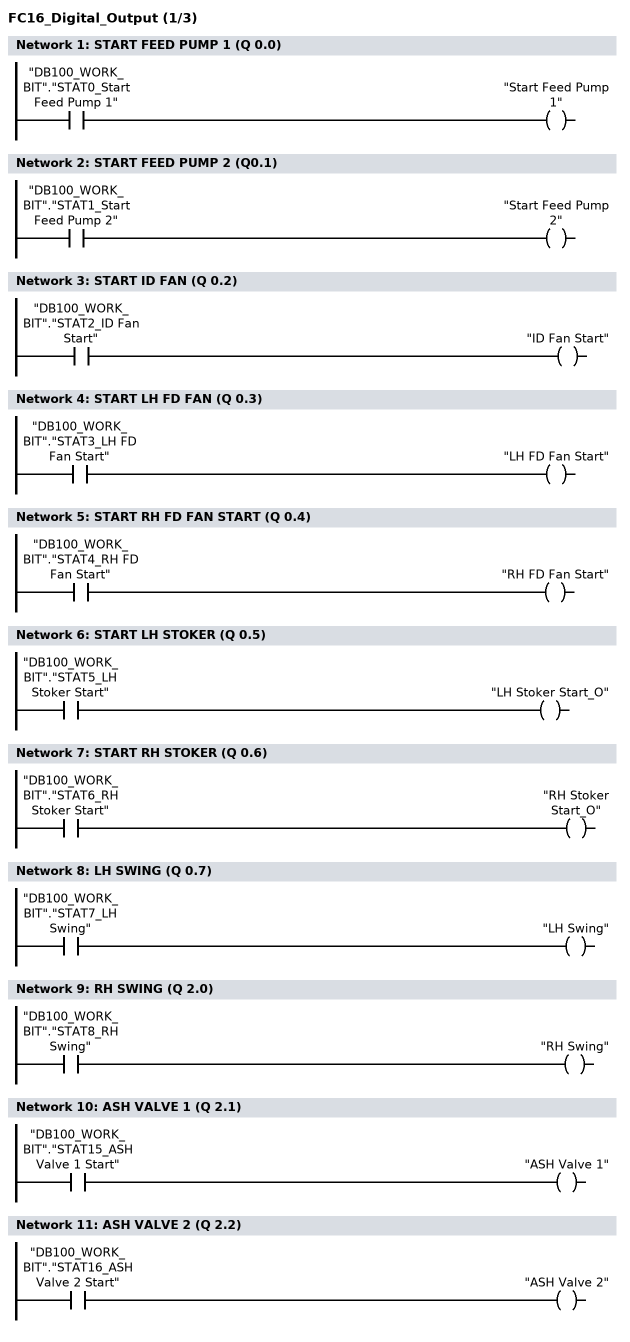
   RUNG wire#powerrail
      Contact( "DB100_WORK_BIT"."STAT0_Start Feed Pump 1" )
      Coil( "Start Feed Pump 1" )
   END_RUNG
   // the same network as SCL:
   "Start Feed Pump 1" := "DB100_WORK_BIT"."STAT0_Start Feed Pump 1";
END_REGION

REGION Network 2: START FEED PUMP 2 (Q0.1)
   RUNG wire#powerrail
      Contact( "DB100_WORK_BIT"."STAT1_Start Feed Pump 2" )
      Coil( "Start Feed Pump 2" )
   END_RUNG
   // the same network as SCL:
   "Start Feed Pump 2" := "DB100_WORK_BIT"."STAT1_Start Feed Pump 2";
END_REGION

REGION Network 3: START ID FAN (Q 0.2)
   RUNG wire#powerrail
      Contact( "DB100_WORK_BIT"."STAT2_ID Fan Start" )
      Coil( "ID Fan Start" )
   END_RUNG
   // the same network as SCL:
   "ID Fan Start" := "DB100_WORK_BIT"."STAT2_ID Fan Start";
END_REGION

REGION Network 4: START LH FD FAN (Q 0.3)
   RUNG wire#powerrail
      Contact( "DB100_WORK_BIT"."STAT3_LH FD Fan Start" )
      Coil( "LH FD Fan Start" )
   END_RUNG
   // the same network as SCL:
   "LH FD Fan Start" := "DB100_WORK_BIT"."STAT3_LH FD Fan Start";
END_REGION

REGION Network 5: START RH FD FAN START (Q 0.4)
   RUNG wire#powerrail
      Contact( "DB100_WORK_BIT"."STAT4_RH FD Fan Start" )
      Coil( "RH FD Fan Start" )
   END_RUNG
   // the same network as SCL:
   "RH FD Fan Start" := "DB100_WORK_BIT"."STAT4_RH FD Fan Start";
END_REGION

REGION Network 6: START LH STOKER (Q 0.5)
   RUNG wire#powerrail
      Contact( "DB100_WORK_BIT"."STAT5_LH Stoker Start" )
      Coil( "LH Stoker Start_O" )
   END_RUNG
   // the same network as SCL:
   "LH Stoker Start_O" := "DB100_WORK_BIT"."STAT5_LH Stoker Start";
END_REGION

REGION Network 7: START RH STOKER (Q 0.6)
   RUNG wire#powerrail
      Contact( "DB100_WORK_BIT"."STAT6_RH Stoker Start" )
      Coil( "RH Stoker Start_O" )
   END_RUNG
   // the same network as SCL:
   "RH Stoker Start_O" := "DB100_WORK_BIT"."STAT6_RH Stoker Start";
END_REGION

REGION Network 8: LH SWING (Q 0.7)
   RUNG wire#powerrail
      Contact( "DB100_WORK_BIT"."STAT7_LH Swing" )
      Coil( "LH Swing" )
   END_RUNG
   // the same network as SCL:
   "LH Swing" := "DB100_WORK_BIT"."STAT7_LH Swing";
END_REGION

REGION Network 9: RH SWING (Q 2.0)
   RUNG wire#powerrail
      Contact( "DB100_WORK_BIT"."STAT8_RH Swing" )
      Coil( "RH Swing" )
   END_RUNG
   // the same network as SCL:
   "RH Swing" := "DB100_WORK_BIT"."STAT8_RH Swing";
END_REGION

REGION Network 10: ASH VALVE 1 (Q 2.1)
   RUNG wire#powerrail
      Contact( "DB100_WORK_BIT"."STAT15_ASH Valve 1 Start" )
      Coil( "ASH Valve 1" )
   END_RUNG
   // the same network as SCL:
   "ASH Valve 1" := "DB100_WORK_BIT"."STAT15_ASH Valve 1 Start";
END_REGION

REGION Network 11: ASH VALVE 2 (Q 2.2)
   RUNG wire#powerrail
      Contact( "DB100_WORK_BIT"."STAT16_ASH Valve 2 Start" )
      Coil( "ASH Valve 2" )
   END_RUNG
   // the same network as SCL:
   "ASH Valve 2" := "DB100_WORK_BIT"."STAT16_ASH Valve 2 Start";
END_REGION

REGION Network 12: ASH CONVEYOR (Q 2.3)
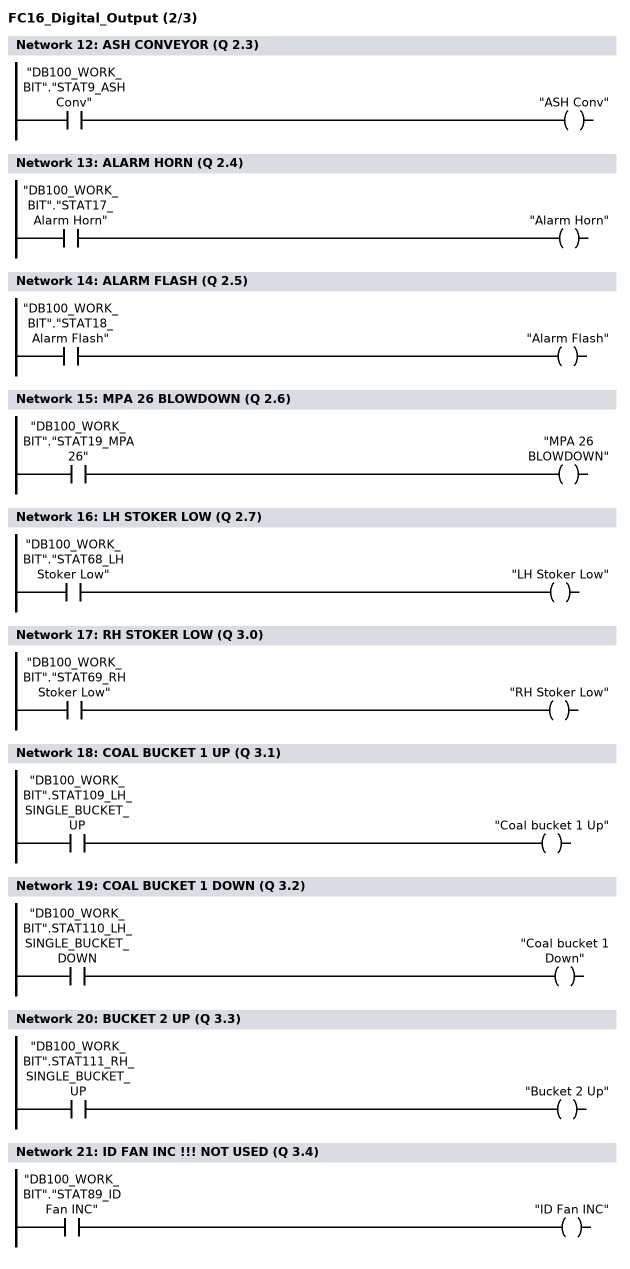
   RUNG wire#powerrail
      Contact( "DB100_WORK_BIT"."STAT9_ASH Conv" )
      Coil( "ASH Conv" )
   END_RUNG
   // the same network as SCL:
   "ASH Conv" := "DB100_WORK_BIT"."STAT9_ASH Conv";
END_REGION

REGION Network 13: ALARM HORN (Q 2.4)
   RUNG wire#powerrail
      Contact( "DB100_WORK_BIT"."STAT17_Alarm Horn" )
      Coil( "Alarm Horn" )
   END_RUNG
   // the same network as SCL:
   "Alarm Horn" := "DB100_WORK_BIT"."STAT17_Alarm Horn";
END_REGION

REGION Network 14: ALARM FLASH (Q 2.5)
   RUNG wire#powerrail
      Contact( "DB100_WORK_BIT"."STAT18_Alarm Flash" )
      Coil( "Alarm Flash" )
   END_RUNG
   // the same network as SCL:
   "Alarm Flash" := "DB100_WORK_BIT"."STAT18_Alarm Flash";
END_REGION

REGION Network 15: MPA 26 BLOWDOWN (Q 2.6)
   RUNG wire#powerrail
      Contact( "DB100_WORK_BIT"."STAT19_MPA 26" )
      Coil( "MPA 26 BLOWDOWN" )
   END_RUNG
   // the same network as SCL:
   "MPA 26 BLOWDOWN" := "DB100_WORK_BIT"."STAT19_MPA 26";
END_REGION

REGION Network 16: LH STOKER LOW (Q 2.7)
   RUNG wire#powerrail
      Contact( "DB100_WORK_BIT"."STAT68_LH Stoker Low" )
      Coil( "LH Stoker Low" )
   END_RUNG
   // the same network as SCL:
   "LH Stoker Low" := "DB100_WORK_BIT"."STAT68_LH Stoker Low";
END_REGION

REGION Network 17: RH STOKER LOW (Q 3.0)
   RUNG wire#powerrail
      Contact( "DB100_WORK_BIT"."STAT69_RH Stoker Low" )
      Coil( "RH Stoker Low" )
   END_RUNG
   // the same network as SCL:
   "RH Stoker Low" := "DB100_WORK_BIT"."STAT69_RH Stoker Low";
END_REGION

REGION Network 18: COAL BUCKET 1 UP (Q 3.1)
   RUNG wire#powerrail
      Contact( "DB100_WORK_BIT".STAT109_LH_SINGLE_BUCKET_UP )
      Coil( "Coal bucket 1 Up" )
   END_RUNG
   // the same network as SCL:
   "Coal bucket 1 Up" := "DB100_WORK_BIT".STAT109_LH_SINGLE_BUCKET_UP;
END_REGION

REGION Network 19: COAL BUCKET 1 DOWN (Q 3.2)
   RUNG wire#powerrail
      Contact( "DB100_WORK_BIT".STAT110_LH_SINGLE_BUCKET_DOWN )
      Coil( "Coal bucket 1 Down" )
   END_RUNG
   // the same network as SCL:
   "Coal bucket 1 Down" := "DB100_WORK_BIT".STAT110_LH_SINGLE_BUCKET_DOWN;
END_REGION

REGION Network 20: BUCKET 2 UP (Q 3.3)
   RUNG wire#powerrail
      Contact( "DB100_WORK_BIT".STAT111_RH_SINGLE_BUCKET_UP )
      Coil( "Bucket 2 Up" )
   END_RUNG
   // the same network as SCL:
   "Bucket 2 Up" := "DB100_WORK_BIT".STAT111_RH_SINGLE_BUCKET_UP;
END_REGION

REGION Network 21: ID FAN INC !!! NOT USED (Q 3.4)
   RUNG wire#powerrail
      Contact( "DB100_WORK_BIT"."STAT89_ID Fan INC" )
      Coil( "ID Fan INC" )
   END_RUNG
   // the same network as SCL:
   "ID Fan INC" := "DB100_WORK_BIT"."STAT89_ID Fan INC";
END_REGION

REGION Network 22: ID FAN DEC !!! NOT USED (Q 3.5)
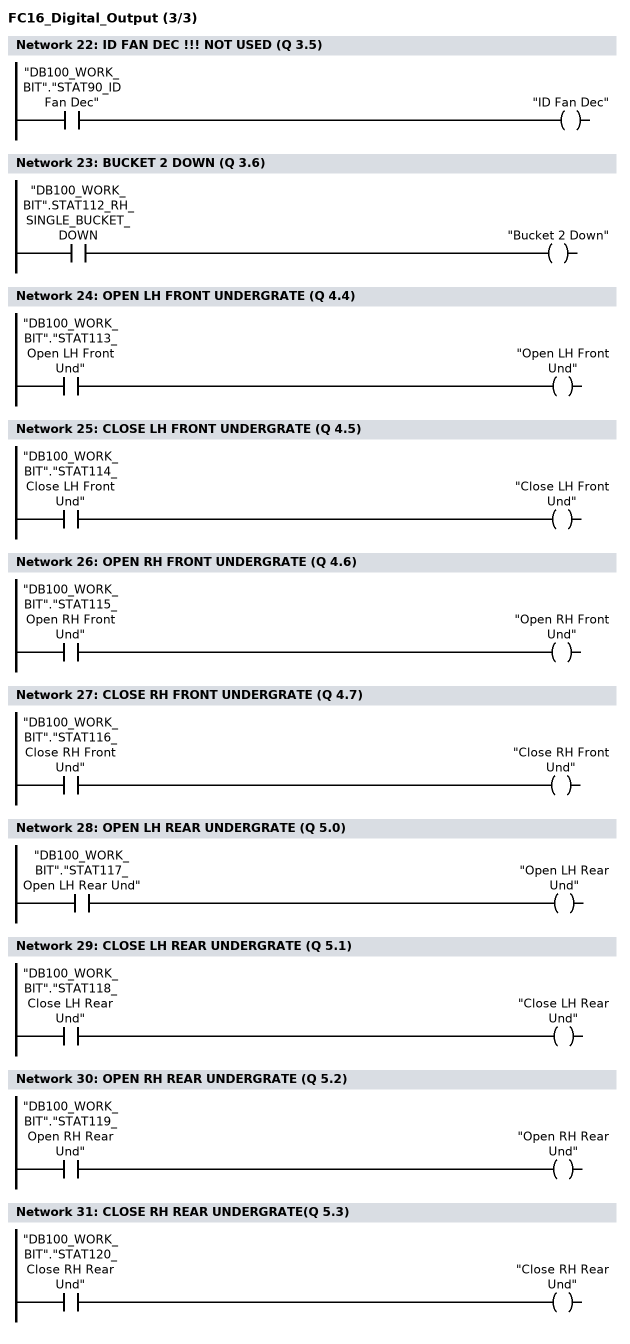
   RUNG wire#powerrail
      Contact( "DB100_WORK_BIT"."STAT90_ID Fan Dec" )
      Coil( "ID Fan Dec" )
   END_RUNG
   // the same network as SCL:
   "ID Fan Dec" := "DB100_WORK_BIT"."STAT90_ID Fan Dec";
END_REGION

REGION Network 23: BUCKET 2 DOWN (Q 3.6)
   RUNG wire#powerrail
      Contact( "DB100_WORK_BIT".STAT112_RH_SINGLE_BUCKET_DOWN )
      Coil( "Bucket 2 Down" )
   END_RUNG
   // the same network as SCL:
   "Bucket 2 Down" := "DB100_WORK_BIT".STAT112_RH_SINGLE_BUCKET_DOWN;
END_REGION

REGION Network 24: OPEN LH FRONT UNDERGRATE (Q 4.4)
   RUNG wire#powerrail
      Contact( "DB100_WORK_BIT"."STAT113_Open LH Front Und" )
      Coil( "Open LH Front Und" )
   END_RUNG
   // the same network as SCL:
   "Open LH Front Und" := "DB100_WORK_BIT"."STAT113_Open LH Front Und";
END_REGION

REGION Network 25: CLOSE LH FRONT UNDERGRATE (Q 4.5)
   RUNG wire#powerrail
      Contact( "DB100_WORK_BIT"."STAT114_Close LH Front Und" )
      Coil( "Close LH Front Und" )
   END_RUNG
   // the same network as SCL:
   "Close LH Front Und" := "DB100_WORK_BIT"."STAT114_Close LH Front Und";
END_REGION

REGION Network 26: OPEN RH FRONT UNDERGRATE (Q 4.6)
   RUNG wire#powerrail
      Contact( "DB100_WORK_BIT"."STAT115_Open RH Front Und" )
      Coil( "Open RH Front Und" )
   END_RUNG
   // the same network as SCL:
   "Open RH Front Und" := "DB100_WORK_BIT"."STAT115_Open RH Front Und";
END_REGION

REGION Network 27: CLOSE RH FRONT UNDERGRATE (Q 4.7)
   RUNG wire#powerrail
      Contact( "DB100_WORK_BIT"."STAT116_Close RH Front Und" )
      Coil( "Close RH Front Und" )
   END_RUNG
   // the same network as SCL:
   "Close RH Front Und" := "DB100_WORK_BIT"."STAT116_Close RH Front Und";
END_REGION

REGION Network 28: OPEN LH REAR UNDERGRATE (Q 5.0)
   RUNG wire#powerrail
      Contact( "DB100_WORK_BIT"."STAT117_Open LH Rear Und" )
      Coil( "Open LH Rear Und" )
   END_RUNG
   // the same network as SCL:
   "Open LH Rear Und" := "DB100_WORK_BIT"."STAT117_Open LH Rear Und";
END_REGION

REGION Network 29: CLOSE LH REAR UNDERGRATE (Q 5.1)
   RUNG wire#powerrail
      Contact( "DB100_WORK_BIT"."STAT118_Close LH Rear Und" )
      Coil( "Close LH Rear Und" )
   END_RUNG
   // the same network as SCL:
   "Close LH Rear Und" := "DB100_WORK_BIT"."STAT118_Close LH Rear Und";
END_REGION

REGION Network 30: OPEN RH REAR UNDERGRATE (Q 5.2)
   RUNG wire#powerrail
      Contact( "DB100_WORK_BIT"."STAT119_Open RH Rear Und" )
      Coil( "Open RH Rear Und" )
   END_RUNG
   // the same network as SCL:
   "Open RH Rear Und" := "DB100_WORK_BIT"."STAT119_Open RH Rear Und";
END_REGION

REGION Network 31: CLOSE RH REAR UNDERGRATE(Q 5.3)
   RUNG wire#powerrail
      Contact( "DB100_WORK_BIT"."STAT120_Close RH Rear Und" )
      Coil( "Close RH Rear Und" )
   END_RUNG
   // the same network as SCL:
   "Close RH Rear Und" := "DB100_WORK_BIT"."STAT120_Close RH Rear Und";
END_REGION
END_FUNCTION

FUNCTION "FC17_Analog_Input" : Void   // FC17, LAD
TITLE = Mapping Analog Input to DB 103
{ S7_Optimized_Access := 'TRUE' }
VERSION : 0.1
BEGIN

REGION Network 1: Pressure Transducer IW 100
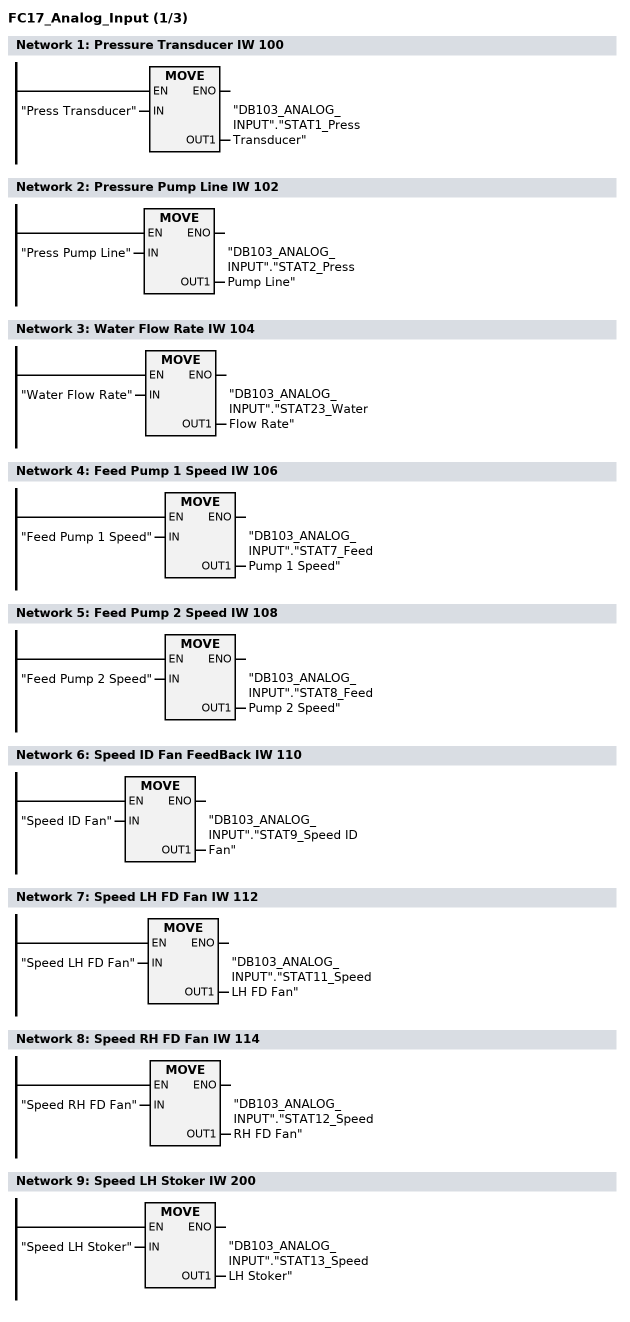
   RUNG wire#powerrail
      Move(in := "Press Transducer", out1 => "DB103_ANALOG_INPUT"."STAT1_Press Transducer")
   END_RUNG
   // the same network as SCL:
   "DB103_ANALOG_INPUT"."STAT1_Press Transducer" := "Press Transducer";
END_REGION

REGION Network 2: Pressure Pump Line IW 102
   RUNG wire#powerrail
      Move(in := "Press Pump Line", out1 => "DB103_ANALOG_INPUT"."STAT2_Press Pump Line")
   END_RUNG
   // the same network as SCL:
   "DB103_ANALOG_INPUT"."STAT2_Press Pump Line" := "Press Pump Line";
END_REGION

REGION Network 3: Water Flow Rate IW 104
   RUNG wire#powerrail
      Move(in := "Water Flow Rate", out1 => "DB103_ANALOG_INPUT"."STAT23_Water Flow Rate")
   END_RUNG
   // the same network as SCL:
   "DB103_ANALOG_INPUT"."STAT23_Water Flow Rate" := "Water Flow Rate";
END_REGION

REGION Network 4: Feed Pump 1 Speed IW 106
   RUNG wire#powerrail
      Move(in := "Feed Pump 1 Speed", out1 => "DB103_ANALOG_INPUT"."STAT7_Feed Pump 1 Speed")
   END_RUNG
   // the same network as SCL:
   "DB103_ANALOG_INPUT"."STAT7_Feed Pump 1 Speed" := "Feed Pump 1 Speed";
END_REGION

REGION Network 5: Feed Pump 2 Speed IW 108
   RUNG wire#powerrail
      Move(in := "Feed Pump 2 Speed", out1 => "DB103_ANALOG_INPUT"."STAT8_Feed Pump 2 Speed")
   END_RUNG
   // the same network as SCL:
   "DB103_ANALOG_INPUT"."STAT8_Feed Pump 2 Speed" := "Feed Pump 2 Speed";
END_REGION

REGION Network 6: Speed ID Fan FeedBack IW 110
   RUNG wire#powerrail
      Move(in := "Speed ID Fan", out1 => "DB103_ANALOG_INPUT"."STAT9_Speed ID Fan")
   END_RUNG
   // the same network as SCL:
   "DB103_ANALOG_INPUT"."STAT9_Speed ID Fan" := "Speed ID Fan";
END_REGION

REGION Network 7: Speed LH FD Fan IW 112
   RUNG wire#powerrail
      Move(in := "Speed LH FD Fan", out1 => "DB103_ANALOG_INPUT"."STAT11_Speed LH FD Fan")
   END_RUNG
   // the same network as SCL:
   "DB103_ANALOG_INPUT"."STAT11_Speed LH FD Fan" := "Speed LH FD Fan";
END_REGION

REGION Network 8: Speed RH FD Fan IW 114
   RUNG wire#powerrail
      Move(in := "Speed RH FD Fan", out1 => "DB103_ANALOG_INPUT"."STAT12_Speed RH FD Fan")
   END_RUNG
   // the same network as SCL:
   "DB103_ANALOG_INPUT"."STAT12_Speed RH FD Fan" := "Speed RH FD Fan";
END_REGION

REGION Network 9: Speed LH Stoker IW 200
   RUNG wire#powerrail
      Move(in := "Speed LH Stoker", out1 => "DB103_ANALOG_INPUT"."STAT13_Speed LH Stoker")
   END_RUNG
   // the same network as SCL:
   "DB103_ANALOG_INPUT"."STAT13_Speed LH Stoker" := "Speed LH Stoker";
END_REGION

REGION Network 10: Speed RH Stoker IW 202
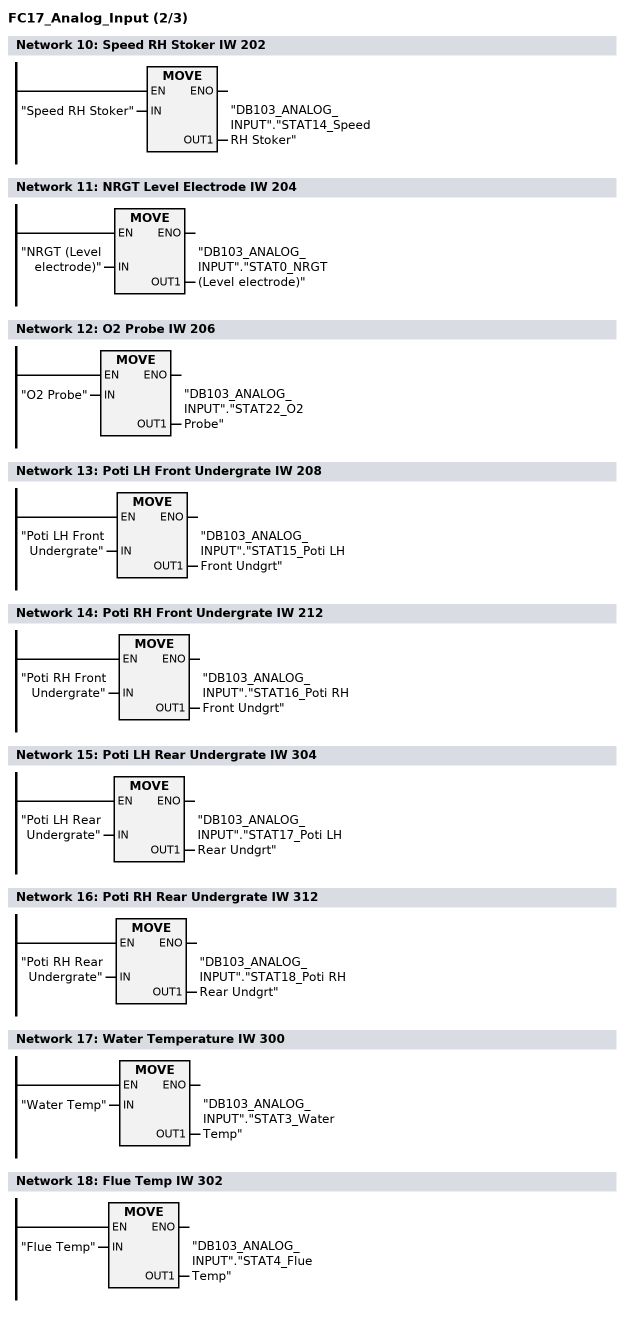
   RUNG wire#powerrail
      Move(in := "Speed RH Stoker", out1 => "DB103_ANALOG_INPUT"."STAT14_Speed RH Stoker")
   END_RUNG
   // the same network as SCL:
   "DB103_ANALOG_INPUT"."STAT14_Speed RH Stoker" := "Speed RH Stoker";
END_REGION

REGION Network 11: NRGT Level Electrode IW 204
   RUNG wire#powerrail
      Move(in := "NRGT (Level electrode)", out1 => "DB103_ANALOG_INPUT"."STAT0_NRGT (Level electrode)")
   END_RUNG
   // the same network as SCL:
   "DB103_ANALOG_INPUT"."STAT0_NRGT (Level electrode)" := "NRGT (Level electrode)";
END_REGION

REGION Network 12: O2 Probe IW 206
   RUNG wire#powerrail
      Move(in := "O2 Probe", out1 => "DB103_ANALOG_INPUT"."STAT22_O2 Probe")
   END_RUNG
   // the same network as SCL:
   "DB103_ANALOG_INPUT"."STAT22_O2 Probe" := "O2 Probe";
END_REGION

REGION Network 13: Poti LH Front Undergrate IW 208
   RUNG wire#powerrail
      Move(in := "Poti LH Front Undergrate", out1 => "DB103_ANALOG_INPUT"."STAT15_Poti LH Front Undgrt")
   END_RUNG
   // the same network as SCL:
   "DB103_ANALOG_INPUT"."STAT15_Poti LH Front Undgrt" := "Poti LH Front Undergrate";
END_REGION

REGION Network 14: Poti RH Front Undergrate IW 212
   RUNG wire#powerrail
      Move(in := "Poti RH Front Undergrate", out1 => "DB103_ANALOG_INPUT"."STAT16_Poti RH Front Undgrt")
   END_RUNG
   // the same network as SCL:
   "DB103_ANALOG_INPUT"."STAT16_Poti RH Front Undgrt" := "Poti RH Front Undergrate";
END_REGION

REGION Network 15: Poti LH Rear Undergrate IW 304
   RUNG wire#powerrail
      Move(in := "Poti LH Rear Undergrate", out1 => "DB103_ANALOG_INPUT"."STAT17_Poti LH Rear Undgrt")
   END_RUNG
   // the same network as SCL:
   "DB103_ANALOG_INPUT"."STAT17_Poti LH Rear Undgrt" := "Poti LH Rear Undergrate";
END_REGION

REGION Network 16: Poti RH Rear Undergrate IW 312
   RUNG wire#powerrail
      Move(in := "Poti RH Rear Undergrate", out1 => "DB103_ANALOG_INPUT"."STAT18_Poti RH Rear Undgrt")
   END_RUNG
   // the same network as SCL:
   "DB103_ANALOG_INPUT"."STAT18_Poti RH Rear Undgrt" := "Poti RH Rear Undergrate";
END_REGION

REGION Network 17: Water Temperature IW 300
   RUNG wire#powerrail
      Move(in := "Water Temp", out1 => "DB103_ANALOG_INPUT"."STAT3_Water Temp")
   END_RUNG
   // the same network as SCL:
   "DB103_ANALOG_INPUT"."STAT3_Water Temp" := "Water Temp";
END_REGION

REGION Network 18: Flue Temp IW 302
   RUNG wire#powerrail
      Move(in := "Flue Temp", out1 => "DB103_ANALOG_INPUT"."STAT4_Flue Temp")
   END_RUNG
   // the same network as SCL:
   "DB103_ANALOG_INPUT"."STAT4_Flue Temp" := "Flue Temp";
END_REGION

REGION Network 19: LH Thermocouple IW 308
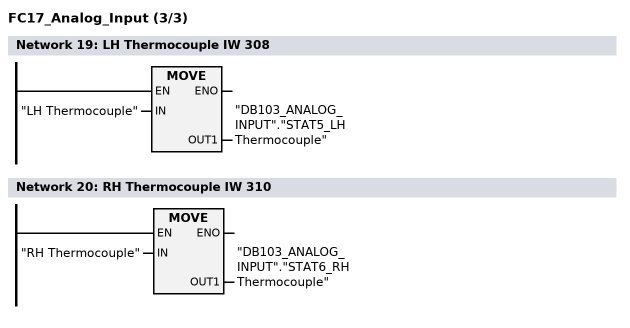
   RUNG wire#powerrail
      Move(in := "LH Thermocouple", out1 => "DB103_ANALOG_INPUT"."STAT5_LH Thermocouple")
   END_RUNG
   // the same network as SCL:
   "DB103_ANALOG_INPUT"."STAT5_LH Thermocouple" := "LH Thermocouple";
END_REGION

REGION Network 20: RH Thermocouple IW 310
   RUNG wire#powerrail
      Move(in := "RH Thermocouple", out1 => "DB103_ANALOG_INPUT"."STAT6_RH Thermocouple")
   END_RUNG
   // the same network as SCL:
   "DB103_ANALOG_INPUT"."STAT6_RH Thermocouple" := "RH Thermocouple";
END_REGION
END_FUNCTION

FUNCTION "FC18_Analog_Output" : Void   // FC18, LAD
TITLE = Mapping Analog Output from DB 140
{ S7_Optimized_Access := 'TRUE' }
VERSION : 0.1
BEGIN

REGION Network 1: Feed Pump 1 Reference Speed QW 500
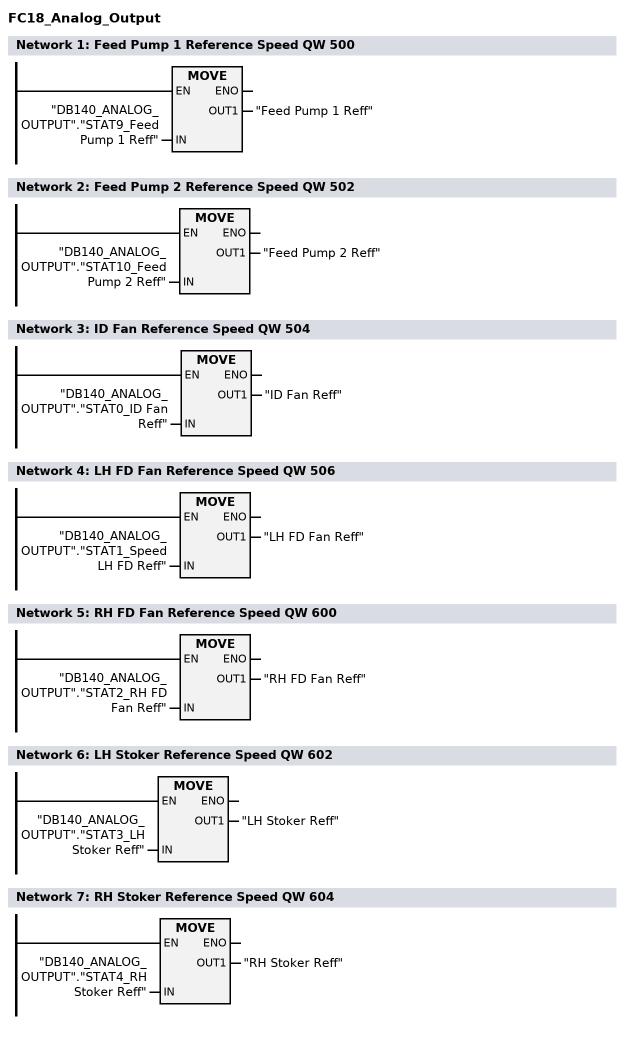
   RUNG wire#powerrail
      Move(in := "DB140_ANALOG_OUTPUT"."STAT9_Feed Pump 1 Reff", out1 => "Feed Pump 1 Reff")
   END_RUNG
   // the same network as SCL:
   "Feed Pump 1 Reff" := "DB140_ANALOG_OUTPUT"."STAT9_Feed Pump 1 Reff";
END_REGION

REGION Network 2: Feed Pump 2 Reference Speed QW 502
   RUNG wire#powerrail
      Move(in := "DB140_ANALOG_OUTPUT"."STAT10_Feed Pump 2 Reff", out1 => "Feed Pump 2 Reff")
   END_RUNG
   // the same network as SCL:
   "Feed Pump 2 Reff" := "DB140_ANALOG_OUTPUT"."STAT10_Feed Pump 2 Reff";
END_REGION

REGION Network 3: ID Fan Reference Speed QW 504
   RUNG wire#powerrail
      Move(in := "DB140_ANALOG_OUTPUT"."STAT0_ID Fan Reff", out1 => "ID Fan Reff")
   END_RUNG
   // the same network as SCL:
   "ID Fan Reff" := "DB140_ANALOG_OUTPUT"."STAT0_ID Fan Reff";
END_REGION

REGION Network 4: LH FD Fan Reference Speed QW 506
   RUNG wire#powerrail
      Move(in := "DB140_ANALOG_OUTPUT"."STAT1_Speed LH FD Reff", out1 => "LH FD Fan Reff")
   END_RUNG
   // the same network as SCL:
   "LH FD Fan Reff" := "DB140_ANALOG_OUTPUT"."STAT1_Speed LH FD Reff";
END_REGION

REGION Network 5: RH FD Fan Reference Speed QW 600
   RUNG wire#powerrail
      Move(in := "DB140_ANALOG_OUTPUT"."STAT2_RH FD Fan Reff", out1 => "RH FD Fan Reff")
   END_RUNG
   // the same network as SCL:
   "RH FD Fan Reff" := "DB140_ANALOG_OUTPUT"."STAT2_RH FD Fan Reff";
END_REGION

REGION Network 6: LH Stoker Reference Speed QW 602
   RUNG wire#powerrail
      Move(in := "DB140_ANALOG_OUTPUT"."STAT3_LH Stoker Reff", out1 => "LH Stoker Reff")
   END_RUNG
   // the same network as SCL:
   "LH Stoker Reff" := "DB140_ANALOG_OUTPUT"."STAT3_LH Stoker Reff";
END_REGION

REGION Network 7: RH Stoker Reference Speed QW 604
   RUNG wire#powerrail
      Move(in := "DB140_ANALOG_OUTPUT"."STAT4_RH Stoker Reff", out1 => "RH Stoker Reff")
   END_RUNG
   // the same network as SCL:
   "RH Stoker Reff" := "DB140_ANALOG_OUTPUT"."STAT4_RH Stoker Reff";
END_REGION
END_FUNCTION

FUNCTION "FC105_scalling AI" : Void   // FC105, LAD
TITLE = SCALLING ANALOG INPUT
{ S7_Optimized_Access := 'TRUE' }
VERSION : 0.1
// rumus scalling
// 
// norm_x  = out =  (VALUE – MIN) / (MAX – MIN)
// scale_x  = out =( (max-min)*value)+min
   VAR_INPUT
      IN0 : Int;
      IN1 : Real;
      IN2 : Real;
      IN3 : Bool;
   END_VAR
   VAR_OUTPUT
      Out4 : Real;
      RET_VAL_1 : Word;
   END_VAR
   VAR_TEMP
      Temp5 : Real;
      Temp6 : Real;
      Temp7 : Real;
      Temp8 : Real;
      Temp9 : Real;
      Temp10 : DInt;
      Temp11 : Bool;
      Temp12 : Bool;
      Temp13 : Real;
      Temp14 : Real;
      Temp15 : Real;
   END_VAR
   VAR_TEMP   // added for the SCL form of the ladder/FBD networks
      _w1 : Bool;
   END_VAR
BEGIN

REGION Network 1: K1 min
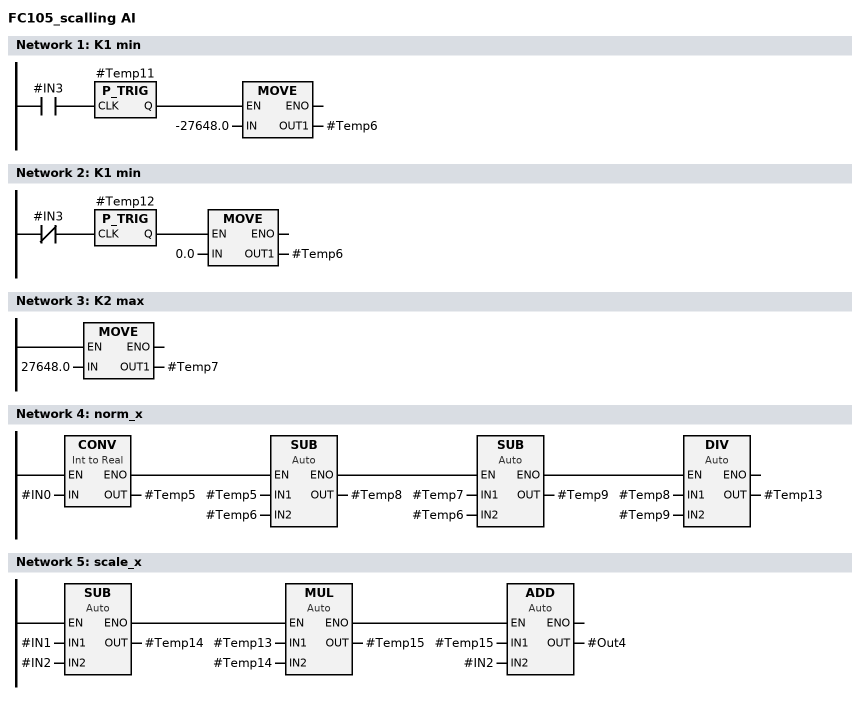
   RUNG wire#powerrail
      Contact( #IN3 )
      P_Trig( #Temp11 )
      Move(in := -27648.0, out1 => #Temp6)
   END_RUNG
   // the same network as SCL:
   #_w1 := #IN3 AND NOT #Temp11;   // rising edge
   #Temp11 := #IN3;
   IF #_w1 THEN #Temp6 := -27648.0; END_IF;
END_REGION

REGION Network 2: K1 min
   RUNG wire#powerrail
      I_Contact( #IN3 )
      P_Trig( #Temp12 )
      Move(in := 0.0, out1 => #Temp6)
   END_RUNG
   // the same network as SCL:
   #_w1 := NOT #IN3 AND NOT #Temp12;   // rising edge
   #Temp12 := NOT #IN3;
   IF #_w1 THEN #Temp6 := 0.0; END_IF;
END_REGION

REGION Network 3: K2 max
   RUNG wire#powerrail
      Move(in := 27648.0, out1 => #Temp7)
   END_RUNG
   // the same network as SCL:
   #Temp7 := 27648.0;
END_REGION

REGION Network 4: norm_x
   RUNG wire#powerrail
      { S7_Templates := "[SrcType := Int, DestType := Real]" } Convert(in := #IN0, out => #Temp5)
      Sub(in1 := #Temp5, in2 := #Temp6, out => #Temp8)
      Sub(in1 := #Temp7, in2 := #Temp6, out => #Temp9)
      Div(in1 := #Temp8, in2 := #Temp9, out => #Temp13)
   END_RUNG
   // the same network as SCL:
   #Temp5 := INT_TO_REAL(#IN0);
   #Temp8 := #Temp5 - #Temp6;
   #Temp9 := #Temp7 - #Temp6;
   #Temp13 := #Temp8 / #Temp9;
END_REGION

REGION Network 5: scale_x
   RUNG wire#powerrail
      Sub(in1 := #IN1, in2 := #IN2, out => #Temp14)
      Mul(in1 := #Temp13, in2 := #Temp14, out => #Temp15)
      Add(in1 := #Temp15, in2 := #IN2, out => #Out4)
   END_RUNG
   // the same network as SCL:
   #Temp14 := #IN1 - #IN2;
   #Temp15 := #Temp13 * #Temp14;
   #Out4 := #Temp15 + #IN2;
END_REGION
END_FUNCTION

FUNCTION "FC106_Unscalling" : Void   // FC106, LAD
TITLE = UNSCALLING
{ S7_Optimized_Access := 'TRUE' }
VERSION : 0.1
// rumus scalling
// 
// norm_x  = out =  (VALUE – MIN) / (MAX – MIN)
// scale_x  = out =( (max-min)*value)+min
   VAR_INPUT
      IN0 : Real;
      IN1 : Real;
      IN2 : Real;
      IN3 : Bool;
   END_VAR
   VAR_OUTPUT
      Out4 : Int;
   END_VAR
   VAR_TEMP
      Temp5 : Real;
      Temp6 : Real;
      Temp7 : Real;
      Temp8 : Real;
      Temp9 : Real;
      Temp10 : Real;
      Temp11 : Bool;
      Temp12 : Bool;
      Temp13 : Real;
      Temp14 : Real;
      Temp15 : Int;
   END_VAR
   VAR_TEMP   // added for the SCL form of the ladder/FBD networks
      _w1 : Bool;
   END_VAR
BEGIN

REGION Network 1: MIN
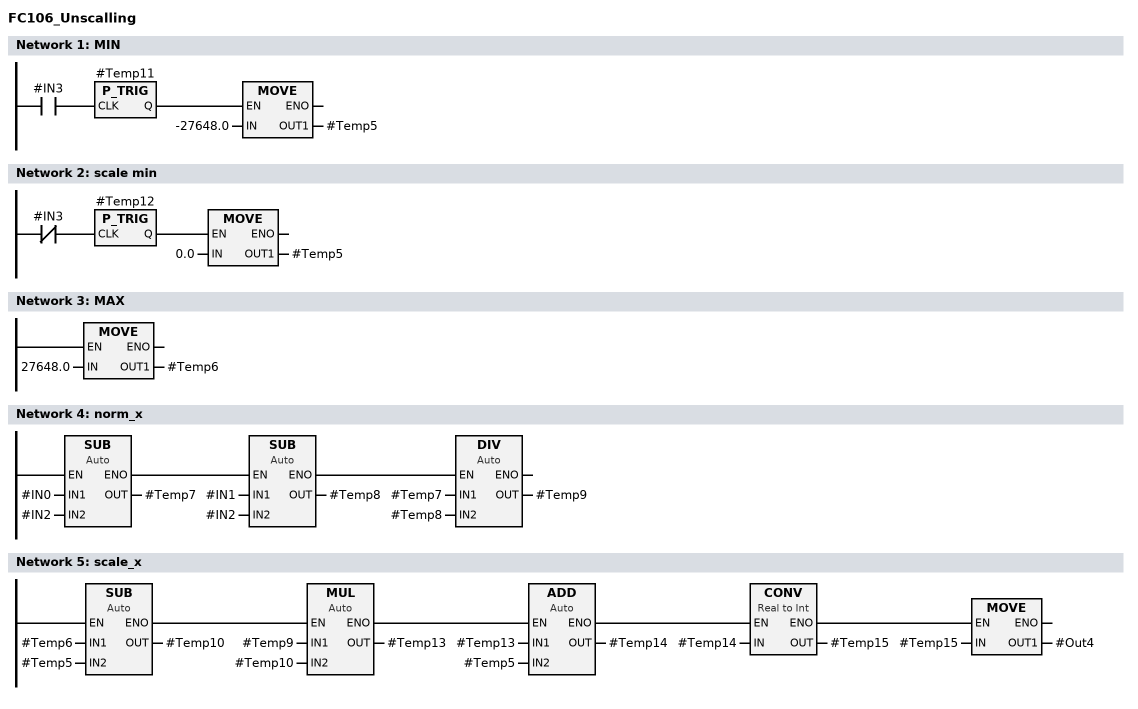
   RUNG wire#powerrail
      Contact( #IN3 )
      P_Trig( #Temp11 )
      Move(in := -27648.0, out1 => #Temp5)
   END_RUNG
   // the same network as SCL:
   #_w1 := #IN3 AND NOT #Temp11;   // rising edge
   #Temp11 := #IN3;
   IF #_w1 THEN #Temp5 := -27648.0; END_IF;
END_REGION

REGION Network 2: scale min
   RUNG wire#powerrail
      I_Contact( #IN3 )
      P_Trig( #Temp12 )
      Move(in := 0.0, out1 => #Temp5)
   END_RUNG
   // the same network as SCL:
   #_w1 := NOT #IN3 AND NOT #Temp12;   // rising edge
   #Temp12 := NOT #IN3;
   IF #_w1 THEN #Temp5 := 0.0; END_IF;
END_REGION

REGION Network 3: MAX
   RUNG wire#powerrail
      Move(in := 27648.0, out1 => #Temp6)
   END_RUNG
   // the same network as SCL:
   #Temp6 := 27648.0;
END_REGION

REGION Network 4: norm_x
   RUNG wire#powerrail
      Sub(in1 := #IN0, in2 := #IN2, out => #Temp7)
      Sub(in1 := #IN1, in2 := #IN2, out => #Temp8)
      Div(in1 := #Temp7, in2 := #Temp8, out => #Temp9)
   END_RUNG
   // the same network as SCL:
   #Temp7 := #IN0 - #IN2;
   #Temp8 := #IN1 - #IN2;
   #Temp9 := #Temp7 / #Temp8;
END_REGION

REGION Network 5: scale_x
   RUNG wire#powerrail
      Sub(in1 := #Temp6, in2 := #Temp5, out => #Temp10)
      Mul(in1 := #Temp9, in2 := #Temp10, out => #Temp13)
      Add(in1 := #Temp13, in2 := #Temp5, out => #Temp14)
      { S7_Templates := "[SrcType := Real, DestType := Int]" } Convert(in := #Temp14, out => #Temp15)
      Move(in := #Temp15, out1 => #Out4)
   END_RUNG
   // the same network as SCL:
   #Temp10 := #Temp6 - #Temp5;
   #Temp13 := #Temp9 * #Temp10;
   #Temp14 := #Temp13 + #Temp5;
   #Temp15 := REAL_TO_INT(#Temp14);
   #Out4 := #Temp15;
END_REGION
END_FUNCTION

FUNCTION "FC108_Unscalling_Custom" : Void   // FC108, LAD
TITLE = UNSCALLING CUSTOM
{ S7_Optimized_Access := 'TRUE' }
VERSION : 0.1
   VAR_INPUT
      IN0 : Real;
      IN1 : Real;
      IN2 : Real;
      IN3 : Bool;
      IN4 : Real;
      IN5 : Real;
   END_VAR
   VAR_OUTPUT
      OUT_4 : Int;
   END_VAR
   VAR_TEMP
      TEMP_7 : Int;
      TEMP_8 : Int;
      TEMP_9 : Real;
   END_VAR
BEGIN

REGION Network 1: IN4 = MIN , IN5 = MAX
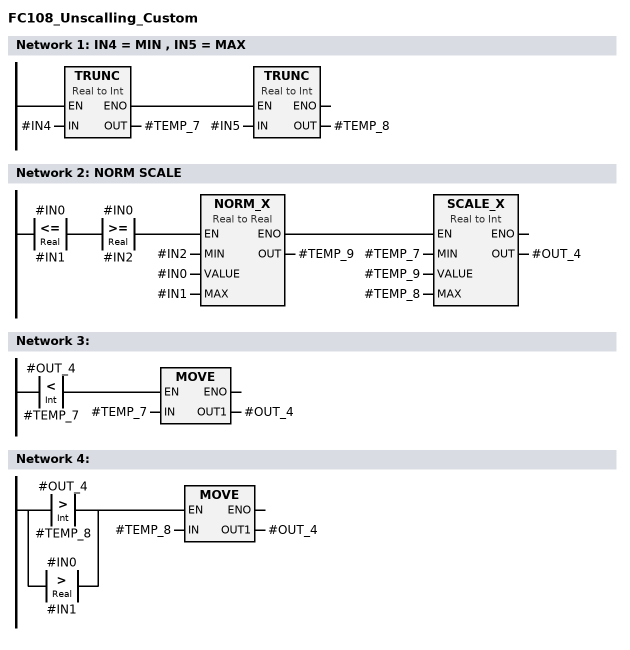
   RUNG wire#powerrail
      { S7_Templates := "[SrcType := Real, DestType := Int]" } Trunc(in := #IN4, out => #TEMP_7)
      { S7_Templates := "[SrcType := Real, DestType := Int]" } Trunc(in := #IN5, out => #TEMP_8)
   END_RUNG
   // the same network as SCL:
   #TEMP_7 := TRUNC(#IN4);
   #TEMP_8 := TRUNC(#IN5);
END_REGION

REGION Network 2: NORM SCALE
   RUNG wire#powerrail
      { S7_Templates := "SrcType := Real" } LE_Contact(in1 := #IN0, in2 := #IN1)
      { S7_Templates := "SrcType := Real" } GE_Contact(in1 := #IN0, in2 := #IN2)
      { S7_Templates := "[SrcType := Real, DestType := Real]" } Normalize(min := #IN2, value := #IN0, max := #IN1, out => #TEMP_9)
      { S7_Templates := "[SrcType := Real, DestType := Int]" } Scale(min := #TEMP_7, value := #TEMP_9, max := #TEMP_8, out => #OUT_4)
   END_RUNG
   // the same network as SCL:
   IF (#IN0 <= #IN1) AND (#IN0 >= #IN2) THEN
       #TEMP_9 := NORM_X(MIN := #IN2, VALUE := #IN0, MAX := #IN1);
       #OUT_4 := SCALE_X(MIN := #TEMP_7, VALUE := #TEMP_9, MAX := #TEMP_8);
   END_IF;
END_REGION

REGION Network 3
   RUNG wire#powerrail
      { S7_Templates := "SrcType := Int" } LT_Contact(in1 := #OUT_4, in2 := #TEMP_7)
      Move(in := #TEMP_7, out1 => #OUT_4)
   END_RUNG
   // the same network as SCL:
   IF #OUT_4 < #TEMP_7 THEN #OUT_4 := #TEMP_7; END_IF;
END_REGION

REGION Network 4
   RUNG wire#powerrail
      { S7_Templates := "SrcType := Int" } GT_Contact(in1 := #OUT_4, in2 := #TEMP_8)
      wire#w1
      Move(in := #TEMP_8, out1 => #OUT_4)
   END_RUNG
   RUNG wire#powerrail
      { S7_Templates := "SrcType := Real" } GT_Contact(in1 := #IN0, in2 := #IN1)
   END_RUNG wire#w1
   // the same network as SCL:
   IF (#OUT_4 > #TEMP_8) OR (#IN0 > #IN1) THEN #OUT_4 := #TEMP_8; END_IF;
END_REGION
END_FUNCTION

FUNCTION "FC109_Scalling_AI_Custom" : Void   // FC109, LAD
TITLE = SCALLING AI CUSTOM
{ S7_Optimized_Access := 'TRUE' }
VERSION : 0.1
// For analog in undergrate damper
   VAR_INPUT
      IN0 : Int;
      IN1 : Real;
      IN2 : Real;
      IN3 : Bool;
      IN4 : Real;
      IN5 : Real;
   END_VAR
   VAR_OUTPUT
      Out4 : Real;
      RET_VAL_1 : Word;
   END_VAR
   VAR_TEMP
      TEMP_8 : Int;
      TEMP_7 : Int;
      TEMP_9 : Real;
      TEMP_10 : Real;
   END_VAR
BEGIN

REGION Network 1: convert integer to real
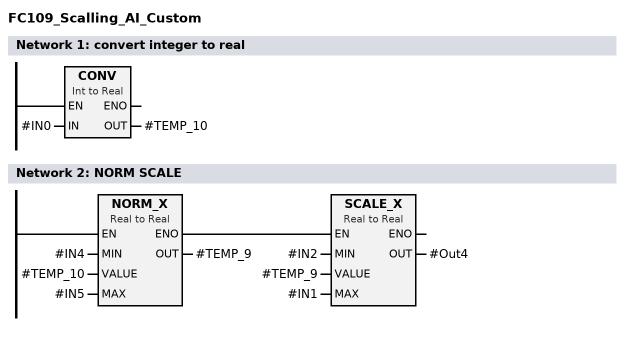
   RUNG wire#powerrail
      { S7_Templates := "[SrcType := Int, DestType := Real]" } Convert(in := #IN0, out => #TEMP_10)
   END_RUNG
   // the same network as SCL:
   #TEMP_10 := INT_TO_REAL(#IN0);
END_REGION

REGION Network 2: NORM SCALE
   RUNG wire#powerrail
      { S7_Templates := "[SrcType := Real, DestType := Real]" } Normalize(min := #IN4, value := #TEMP_10, max := #IN5, out => #TEMP_9)
      { S7_Templates := "[SrcType := Real, DestType := Real]" } Scale(min := #IN2, value := #TEMP_9, max := #IN1, out => #Out4)
   END_RUNG
   // the same network as SCL:
   #TEMP_9 := NORM_X(MIN := #IN4, VALUE := #TEMP_10, MAX := #IN5);
   #Out4 := SCALE_X(MIN := #IN2, VALUE := #TEMP_9, MAX := #IN1);
END_REGION
END_FUNCTION

FUNCTION "FC110_GENERAL_BIT" : Void   // FC110, LAD
{ S7_Optimized_Access := 'TRUE' }
VERSION : 0.1
BEGIN

REGION Network 1: Always TRUE
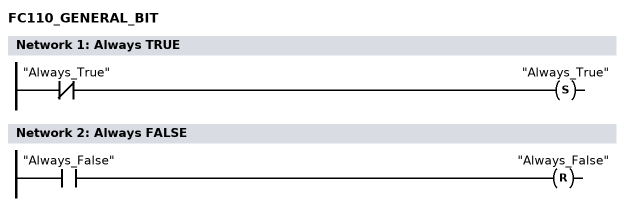
   RUNG wire#powerrail
      I_Contact( "Always_True" )
      S_Coil( "Always_True" )
   END_RUNG
   // the same network as SCL:
   IF NOT "Always_True" THEN "Always_True" := TRUE; END_IF;
END_REGION

REGION Network 2: Always FALSE
   RUNG wire#powerrail
      Contact( "Always_False" )
      R_Coil( "Always_False" )
   END_RUNG
   // the same network as SCL:
   IF "Always_False" THEN "Always_False" := FALSE; END_IF;
END_REGION
END_FUNCTION

FUNCTION "FC112_DATE_TIME" : Void   // FC112, LAD
TITLE = DATE TIME PLC SETTING
{ S7_Optimized_Access := 'TRUE' }
VERSION : 0.1
   VAR_TEMP
      v1 : Int;
      v2 : Word;
      v3 : Int;
      v4 : Word;
      v5 : Int;
      v6 : Word;
      v7 : Int;
      v8 : Word;
      v9 : Int;
      v10 : String;
      v11 : String;
      v12 : Int;
      v13 : Int;
      v14 : Word;
      v15 : Int;
      v16 : Word;
      v17 : Int;
      v18 : Word;
   END_VAR
   VAR_TEMP   // added for the SCL form of the ladder/FBD networks
      _w1 : Bool;
   END_VAR
BEGIN

REGION Network 1: READ DATE TIME
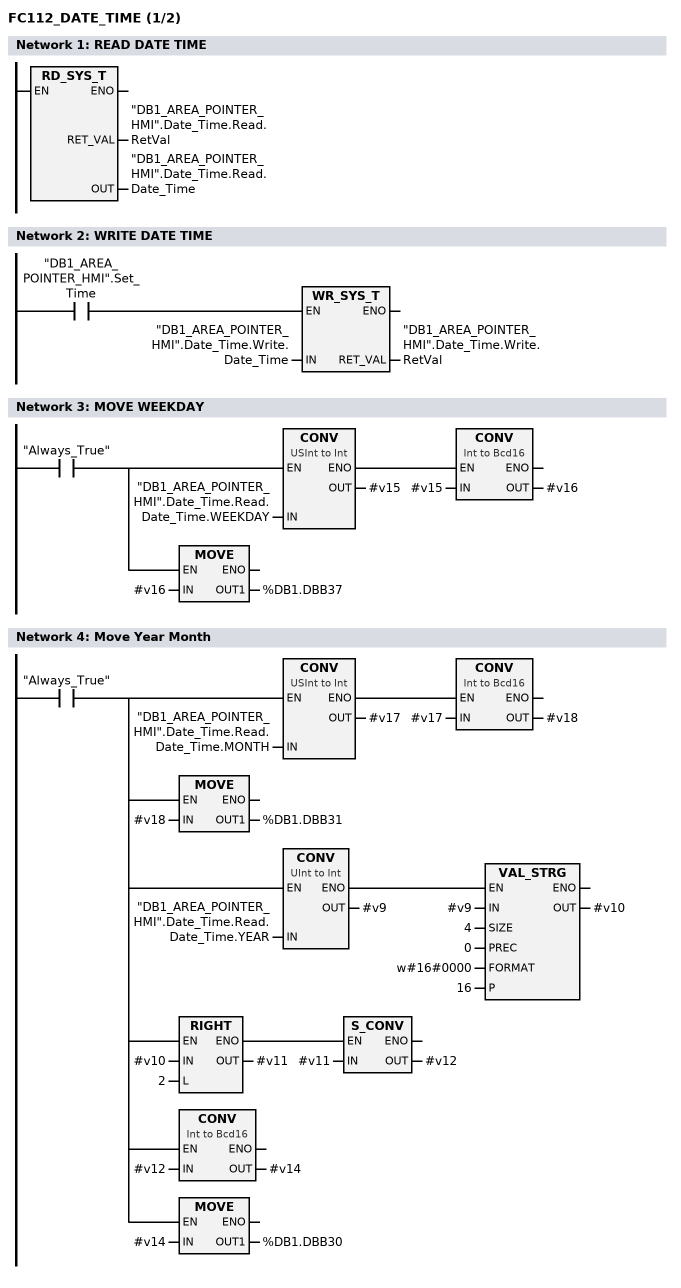
   "DB1_AREA_POINTER_HMI".Date_Time.Read.RetVal := RD_SYS_T(OUT => "DB1_AREA_POINTER_HMI".Date_Time.Read.Date_Time);
END_REGION

REGION Network 2: WRITE DATE TIME
   IF "DB1_AREA_POINTER_HMI".Set_Time THEN
       "DB1_AREA_POINTER_HMI".Date_Time.Write.RetVal := WR_SYS_T(IN := "DB1_AREA_POINTER_HMI".Date_Time.Write.Date_Time);
   END_IF;
END_REGION

REGION Network 3: MOVE WEEKDAY
   RUNG wire#powerrail
      Contact( "Always_True" )
      wire#w1
      { S7_Templates := "[SrcType := USInt, DestType := Int]" } Convert(in := "DB1_AREA_POINTER_HMI".Date_Time.Read.Date_Time.WEEKDAY, out => #v15)
      { S7_Templates := "[SrcType := Int, DestType := Bcd16]" } Convert(in := #v15, out => #v16)
   END_RUNG
   RUNG wire#w1
      Move(in := #v16, out1 => %DB1.DBB37)
   END_RUNG
   // the same network as SCL:
   IF "Always_True" THEN
       #v15 := USINT_TO_INT("DB1_AREA_POINTER_HMI".Date_Time.Read.Date_Time.WEEKDAY);
       #v16 := INT_TO_BCD16(#v15);
       %DB1.DBB37 := #v16;
   END_IF;
END_REGION

REGION Network 4: Move Year Month
   IF "Always_True" THEN
       #v17 := USINT_TO_INT("DB1_AREA_POINTER_HMI".Date_Time.Read.Date_Time.MONTH);
       #v18 := INT_TO_BCD16(#v17);
       %DB1.DBB31 := #v18;
       #v9 := UINT_TO_INT("DB1_AREA_POINTER_HMI".Date_Time.Read.Date_Time.YEAR);
   END_IF;
   #_w1 := "Always_True";
   IF #_w1 THEN
       VAL_STRG(IN := #v9, SIZE := 4, PREC := 0, FORMAT := w#16#0000, P := 16, OUT => #v10);
       #v11 := RIGHT(IN := #v10, L := 2);
       #v12 := S_CONV(IN := #v11);
       #v14 := INT_TO_BCD16(#v12);
       %DB1.DBB30 := #v14;
   END_IF;
END_REGION

REGION Network 5: Move Day &Hour
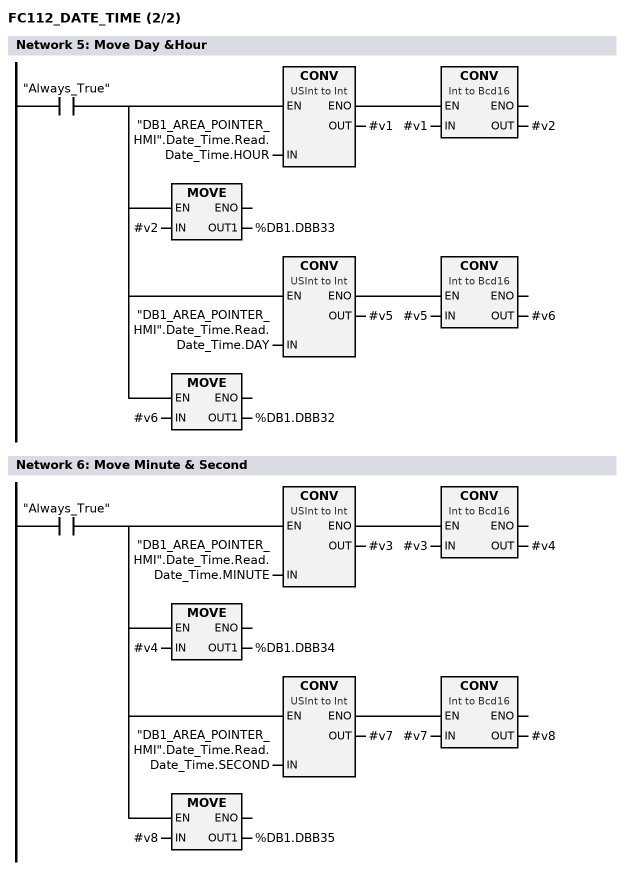
   RUNG wire#powerrail
      Contact( "Always_True" )
      wire#w1
      { S7_Templates := "[SrcType := USInt, DestType := Int]" } Convert(in := "DB1_AREA_POINTER_HMI".Date_Time.Read.Date_Time.HOUR, out => #v1)
      { S7_Templates := "[SrcType := Int, DestType := Bcd16]" } Convert(in := #v1, out => #v2)
   END_RUNG
   RUNG wire#w1
      Move(in := #v2, out1 => %DB1.DBB33)
   END_RUNG
   RUNG wire#w1
      { S7_Templates := "[SrcType := USInt, DestType := Int]" } Convert(in := "DB1_AREA_POINTER_HMI".Date_Time.Read.Date_Time.DAY, out => #v5)
      { S7_Templates := "[SrcType := Int, DestType := Bcd16]" } Convert(in := #v5, out => #v6)
   END_RUNG
   RUNG wire#w1
      Move(in := #v6, out1 => %DB1.DBB32)
   END_RUNG
   // the same network as SCL:
   IF "Always_True" THEN
       #v1 := USINT_TO_INT("DB1_AREA_POINTER_HMI".Date_Time.Read.Date_Time.HOUR);
       #v2 := INT_TO_BCD16(#v1);
       %DB1.DBB33 := #v2;
       #v5 := USINT_TO_INT("DB1_AREA_POINTER_HMI".Date_Time.Read.Date_Time.DAY);
       #v6 := INT_TO_BCD16(#v5);
       %DB1.DBB32 := #v6;
   END_IF;
END_REGION

REGION Network 6: Move Minute & Second
   RUNG wire#powerrail
      Contact( "Always_True" )
      wire#w1
      { S7_Templates := "[SrcType := USInt, DestType := Int]" } Convert(in := "DB1_AREA_POINTER_HMI".Date_Time.Read.Date_Time.MINUTE, out => #v3)
      { S7_Templates := "[SrcType := Int, DestType := Bcd16]" } Convert(in := #v3, out => #v4)
   END_RUNG
   RUNG wire#w1
      Move(in := #v4, out1 => %DB1.DBB34)
   END_RUNG
   RUNG wire#w1
      { S7_Templates := "[SrcType := USInt, DestType := Int]" } Convert(in := "DB1_AREA_POINTER_HMI".Date_Time.Read.Date_Time.SECOND, out => #v7)
      { S7_Templates := "[SrcType := Int, DestType := Bcd16]" } Convert(in := #v7, out => #v8)
   END_RUNG
   RUNG wire#w1
      Move(in := #v8, out1 => %DB1.DBB35)
   END_RUNG
   // the same network as SCL:
   IF "Always_True" THEN
       #v3 := USINT_TO_INT("DB1_AREA_POINTER_HMI".Date_Time.Read.Date_Time.MINUTE);
       #v4 := INT_TO_BCD16(#v3);
       %DB1.DBB34 := #v4;
       #v7 := USINT_TO_INT("DB1_AREA_POINTER_HMI".Date_Time.Read.Date_Time.SECOND);
       #v8 := INT_TO_BCD16(#v7);
       %DB1.DBB35 := #v8;
   END_IF;
END_REGION
END_FUNCTION

ORGANIZATION_BLOCK "Main"   // OB1, LAD, ProgramCycle
TITLE = "Main Program Sweep (Cycle)"
{ S7_Optimized_Access := 'TRUE' }
VERSION : 0.1
   VAR_INPUT
      Initial_Call : Bool;   // Initial call of this OB
      Remanence : Bool;   // =True, if remanent data are available
   END_VAR
BEGIN

REGION Network 1: SCALLING
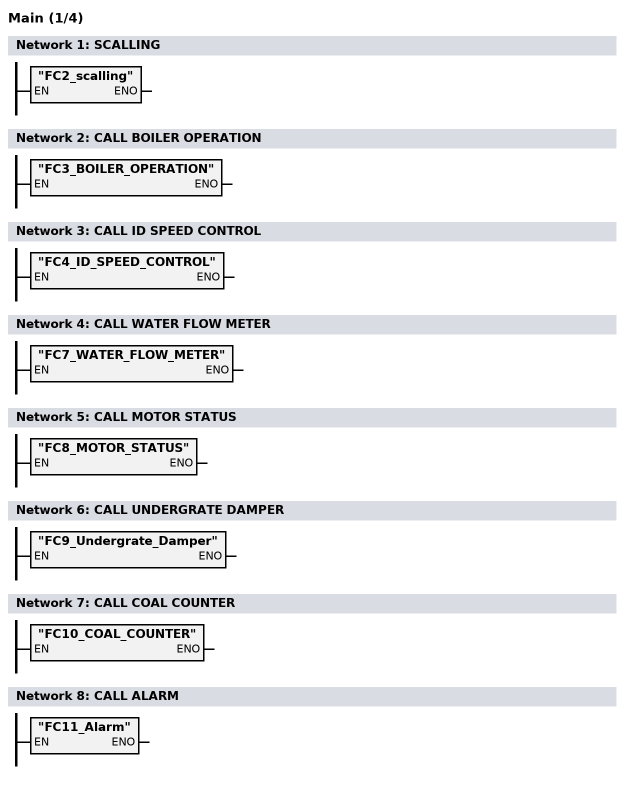
   RUNG wire#powerrail
      "FC2_scalling"()
   END_RUNG
   // the same network as SCL:
   "FC2_scalling"();
END_REGION

REGION Network 2: CALL BOILER OPERATION
   RUNG wire#powerrail
      "FC3_BOILER_OPERATION"()
   END_RUNG
   // the same network as SCL:
   "FC3_BOILER_OPERATION"();
END_REGION

REGION Network 3: CALL ID SPEED CONTROL
   RUNG wire#powerrail
      "FC4_ID_SPEED_CONTROL"()
   END_RUNG
   // the same network as SCL:
   "FC4_ID_SPEED_CONTROL"();
END_REGION

REGION Network 4: CALL WATER FLOW METER
   RUNG wire#powerrail
      "FC7_WATER_FLOW_METER"()
   END_RUNG
   // the same network as SCL:
   "FC7_WATER_FLOW_METER"();
END_REGION

REGION Network 5: CALL MOTOR STATUS
   RUNG wire#powerrail
      "FC8_MOTOR_STATUS"()
   END_RUNG
   // the same network as SCL:
   "FC8_MOTOR_STATUS"();
END_REGION

REGION Network 6: CALL UNDERGRATE DAMPER
   RUNG wire#powerrail
      "FC9_Undergrate_Damper"()
   END_RUNG
   // the same network as SCL:
   "FC9_Undergrate_Damper"();
END_REGION

REGION Network 7: CALL COAL COUNTER
   RUNG wire#powerrail
      "FC10_COAL_COUNTER"()
   END_RUNG
   // the same network as SCL:
   "FC10_COAL_COUNTER"();
END_REGION

REGION Network 8: CALL ALARM
   RUNG wire#powerrail
      "FC11_Alarm"()
   END_RUNG
   // the same network as SCL:
   "FC11_Alarm"();
END_REGION

REGION Network 9: LH SINGLE BUCKET == > FB 5
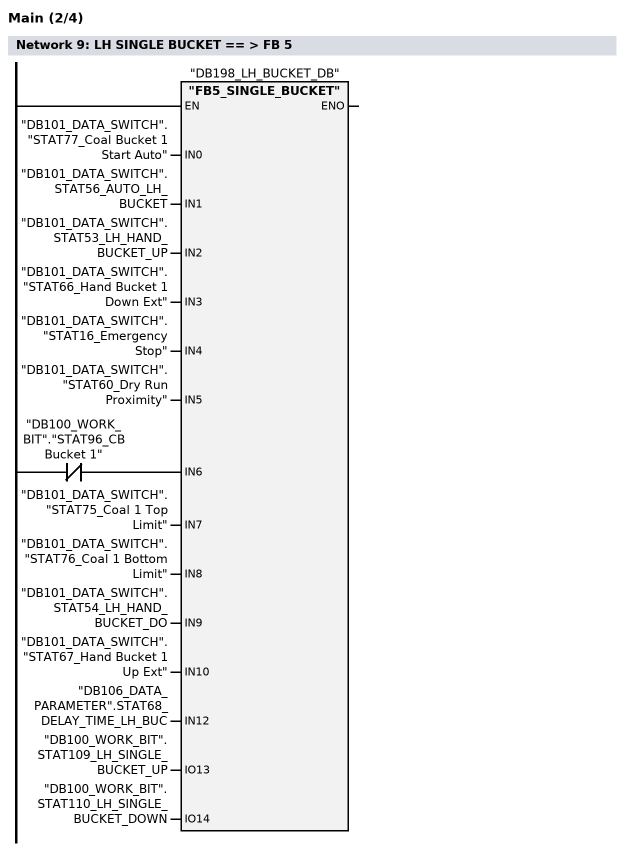
   RUNG wire#powerrail
      "DB198_LH_BUCKET_DB"(IN6 := wire#w1, IN0 := "DB101_DATA_SWITCH"."STAT77_Coal Bucket 1 Start Auto", IN1 := "DB101_DATA_SWITCH".STAT56_AUTO_LH_BUCKET, IN2 := "DB101_DATA_SWITCH".STAT53_LH_HAND_BUCKET_UP, IN3 := "DB101_DATA_SWITCH"."STAT66_Hand Bucket 1 Down Ext", IN4 := "DB101_DATA_SWITCH"."STAT16_Emergency Stop", IN5 := "DB101_DATA_SWITCH"."STAT60_Dry Run Proximity", IN7 := "DB101_DATA_SWITCH"."STAT75_Coal 1 Top Limit", IN8 := "DB101_DATA_SWITCH"."STAT76_Coal 1 Bottom Limit", IN9 := "DB101_DATA_SWITCH".STAT54_LH_HAND_BUCKET_DO, IN10 := "DB101_DATA_SWITCH"."STAT67_Hand Bucket 1 Up Ext", IN12 := "DB106_DATA_PARAMETER".STAT68_DELAY_TIME_LH_BUC, IO13 := "DB100_WORK_BIT".STAT109_LH_SINGLE_BUCKET_UP, IO14 := "DB100_WORK_BIT".STAT110_LH_SINGLE_BUCKET_DOWN)
   END_RUNG
   RUNG wire#powerrail
      I_Contact( "DB100_WORK_BIT"."STAT96_CB Bucket 1" )
   END_RUNG wire#w1
   // the same network as SCL:
   "DB198_LH_BUCKET_DB"(IN0 := "DB101_DATA_SWITCH"."STAT77_Coal Bucket 1 Start Auto",   // "FB5_SINGLE_BUCKET"
                        IN1 := "DB101_DATA_SWITCH".STAT56_AUTO_LH_BUCKET,
                        IN2 := "DB101_DATA_SWITCH".STAT53_LH_HAND_BUCKET_UP,
                        IN3 := "DB101_DATA_SWITCH"."STAT66_Hand Bucket 1 Down Ext",
                        IN4 := "DB101_DATA_SWITCH"."STAT16_Emergency Stop",
                        IN5 := "DB101_DATA_SWITCH"."STAT60_Dry Run Proximity",
                        IN6 := NOT "DB100_WORK_BIT"."STAT96_CB Bucket 1",
                        IN7 := "DB101_DATA_SWITCH"."STAT75_Coal 1 Top Limit",
                        IN8 := "DB101_DATA_SWITCH"."STAT76_Coal 1 Bottom Limit",
                        IN9 := "DB101_DATA_SWITCH".STAT54_LH_HAND_BUCKET_DO,
                        IN10 := "DB101_DATA_SWITCH"."STAT67_Hand Bucket 1 Up Ext",
                        IN12 := "DB106_DATA_PARAMETER".STAT68_DELAY_TIME_LH_BUC,
                        IO13 := "DB100_WORK_BIT".STAT109_LH_SINGLE_BUCKET_UP,
                        IO14 := "DB100_WORK_BIT".STAT110_LH_SINGLE_BUCKET_DOWN);
END_REGION

REGION Network 10: RH SINGLE BUCKET == > FB 5
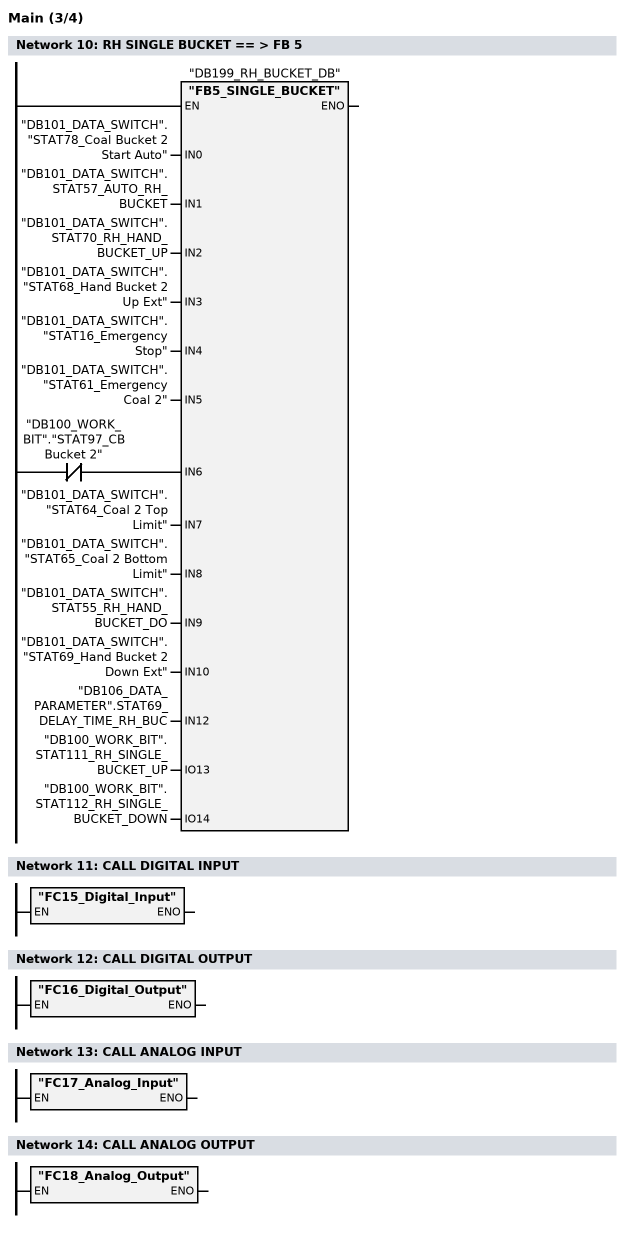
   RUNG wire#powerrail
      "DB199_RH_BUCKET_DB"(IN6 := wire#w1, IN0 := "DB101_DATA_SWITCH"."STAT78_Coal Bucket 2 Start Auto", IN1 := "DB101_DATA_SWITCH".STAT57_AUTO_RH_BUCKET, IN2 := "DB101_DATA_SWITCH".STAT70_RH_HAND_BUCKET_UP, IN3 := "DB101_DATA_SWITCH"."STAT68_Hand Bucket 2 Up Ext", IN4 := "DB101_DATA_SWITCH"."STAT16_Emergency Stop", IN5 := "DB101_DATA_SWITCH"."STAT61_Emergency Coal 2", IN7 := "DB101_DATA_SWITCH"."STAT64_Coal 2 Top Limit", IN8 := "DB101_DATA_SWITCH"."STAT65_Coal 2 Bottom Limit", IN9 := "DB101_DATA_SWITCH".STAT55_RH_HAND_BUCKET_DO, IN10 := "DB101_DATA_SWITCH"."STAT69_Hand Bucket 2 Down Ext", IN12 := "DB106_DATA_PARAMETER".STAT69_DELAY_TIME_RH_BUC, IO13 := "DB100_WORK_BIT".STAT111_RH_SINGLE_BUCKET_UP, IO14 := "DB100_WORK_BIT".STAT112_RH_SINGLE_BUCKET_DOWN)
   END_RUNG
   RUNG wire#powerrail
      I_Contact( "DB100_WORK_BIT"."STAT97_CB Bucket 2" )
   END_RUNG wire#w1
   // the same network as SCL:
   "DB199_RH_BUCKET_DB"(IN0 := "DB101_DATA_SWITCH"."STAT78_Coal Bucket 2 Start Auto",   // "FB5_SINGLE_BUCKET"
                        IN1 := "DB101_DATA_SWITCH".STAT57_AUTO_RH_BUCKET,
                        IN2 := "DB101_DATA_SWITCH".STAT70_RH_HAND_BUCKET_UP,
                        IN3 := "DB101_DATA_SWITCH"."STAT68_Hand Bucket 2 Up Ext",
                        IN4 := "DB101_DATA_SWITCH"."STAT16_Emergency Stop",
                        IN5 := "DB101_DATA_SWITCH"."STAT61_Emergency Coal 2",
                        IN6 := NOT "DB100_WORK_BIT"."STAT97_CB Bucket 2",
                        IN7 := "DB101_DATA_SWITCH"."STAT64_Coal 2 Top Limit",
                        IN8 := "DB101_DATA_SWITCH"."STAT65_Coal 2 Bottom Limit",
                        IN9 := "DB101_DATA_SWITCH".STAT55_RH_HAND_BUCKET_DO,
                        IN10 := "DB101_DATA_SWITCH"."STAT69_Hand Bucket 2 Down Ext",
                        IN12 := "DB106_DATA_PARAMETER".STAT69_DELAY_TIME_RH_BUC,
                        IO13 := "DB100_WORK_BIT".STAT111_RH_SINGLE_BUCKET_UP,
                        IO14 := "DB100_WORK_BIT".STAT112_RH_SINGLE_BUCKET_DOWN);
END_REGION

REGION Network 11: CALL DIGITAL INPUT
   RUNG wire#powerrail
      "FC15_Digital_Input"()
   END_RUNG
   // the same network as SCL:
   "FC15_Digital_Input"();
END_REGION

REGION Network 12: CALL DIGITAL OUTPUT
   RUNG wire#powerrail
      "FC16_Digital_Output"()
   END_RUNG
   // the same network as SCL:
   "FC16_Digital_Output"();
END_REGION

REGION Network 13: CALL ANALOG INPUT
   RUNG wire#powerrail
      "FC17_Analog_Input"()
   END_RUNG
   // the same network as SCL:
   "FC17_Analog_Input"();
END_REGION

REGION Network 14: CALL ANALOG OUTPUT
   RUNG wire#powerrail
      "FC18_Analog_Output"()
   END_RUNG
   // the same network as SCL:
   "FC18_Analog_Output"();
END_REGION

REGION Network 15: BLOWDOWN OPERATION
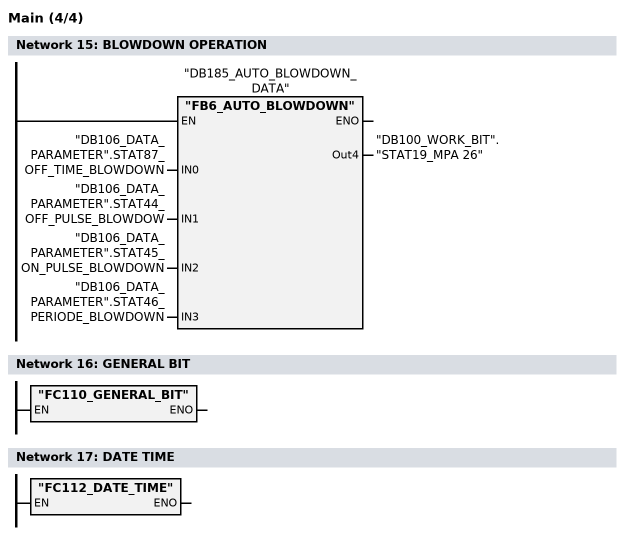
   RUNG wire#powerrail
      "DB185_AUTO_BLOWDOWN_DATA"(IN0 := "DB106_DATA_PARAMETER".STAT87_OFF_TIME_BLOWDOWN, IN1 := "DB106_DATA_PARAMETER".STAT44_OFF_PULSE_BLOWDOW, IN2 := "DB106_DATA_PARAMETER".STAT45_ON_PULSE_BLOWDOWN, IN3 := "DB106_DATA_PARAMETER".STAT46_PERIODE_BLOWDOWN, Out4 => "DB100_WORK_BIT"."STAT19_MPA 26")
   END_RUNG
   // the same network as SCL:
   "DB185_AUTO_BLOWDOWN_DATA"(IN0 := "DB106_DATA_PARAMETER".STAT87_OFF_TIME_BLOWDOWN,   // "FB6_AUTO_BLOWDOWN"
                           IN1 := "DB106_DATA_PARAMETER".STAT44_OFF_PULSE_BLOWDOW,
                           IN2 := "DB106_DATA_PARAMETER".STAT45_ON_PULSE_BLOWDOWN,
                           IN3 := "DB106_DATA_PARAMETER".STAT46_PERIODE_BLOWDOWN,
                           Out4 => "DB100_WORK_BIT"."STAT19_MPA 26");
END_REGION

REGION Network 16: GENERAL BIT
   RUNG wire#powerrail
      "FC110_GENERAL_BIT"()
   END_RUNG
   // the same network as SCL:
   "FC110_GENERAL_BIT"();
END_REGION

REGION Network 17: DATE TIME
   RUNG wire#powerrail
      "FC112_DATE_TIME"()
   END_RUNG
   // the same network as SCL:
   "FC112_DATE_TIME"();
END_REGION
END_ORGANIZATION_BLOCK

ORGANIZATION_BLOCK "Cyclic interrupt"   // OB30, LAD, CyclicInterrupt
{ S7_Optimized_Access := 'TRUE' }
VERSION : 0.1
   VAR_INPUT
      Initial_Call : Bool;   // Initial call of this OB
      Event_Count : Int;   // Events discarded
   END_VAR
BEGIN

REGION Network 1
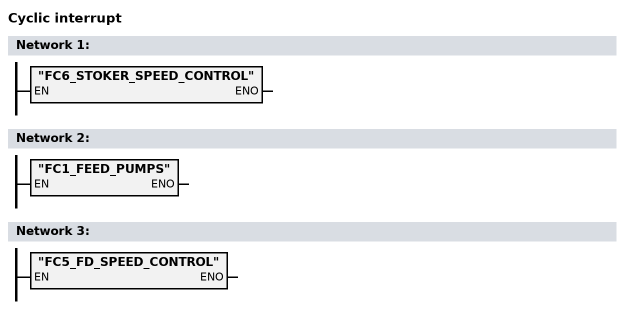
   RUNG wire#powerrail
      "FC6_STOKER_SPEED_CONTROL"()
   END_RUNG
   // the same network as SCL:
   "FC6_STOKER_SPEED_CONTROL"();
END_REGION

REGION Network 2
   RUNG wire#powerrail
      "FC1_FEED_PUMPS"()
   END_RUNG
   // the same network as SCL:
   "FC1_FEED_PUMPS"();
END_REGION

REGION Network 3
   RUNG wire#powerrail
      "FC5_FD_SPEED_CONTROL"()
   END_RUNG
   // the same network as SCL:
   "FC5_FD_SPEED_CONTROL"();
END_REGION
END_ORGANIZATION_BLOCK

ORGANIZATION_BLOCK "OB40"   // OB40, LAD, HWProcessInterrupt
{ S7_Optimized_Access := 'TRUE' }
VERSION : 0.1
   VAR_INPUT
      LADDR : Hw_Io;   // Hardware identifier
      USI : Word;   // User structure identifier
      IChannel : USInt;   // Interrupt channel number
      EventType : Byte;   // EventType
   END_VAR
BEGIN
END_ORGANIZATION_BLOCK

ORGANIZATION_BLOCK "OB80"   // OB80, LAD, TimeErrorInterrupt
{ S7_Optimized_Access := 'TRUE' }
VERSION : 0.1
   VAR_INPUT
      Fault_ID : Byte;   // Fault identifier
      Csg_OBnr : OB_Any;   // Number of OB causing the error
      Csg_Prio : UInt;   // Priority of OB causing the error
   END_VAR
BEGIN
END_ORGANIZATION_BLOCK

ORGANIZATION_BLOCK "OB82"   // OB82, LAD, DiagnosticErrorInterrupt
{ S7_Optimized_Access := 'TRUE' }
VERSION : 0.1
   VAR_INPUT
      IO_State : Word;   // IO state of the HW object
      LADDR : Hw_Any;   // Hardware identifier
      Channel : UInt;   // Channel number
      MultiError : Bool;   // =true if more than one error is present
   END_VAR
BEGIN
END_ORGANIZATION_BLOCK

ORGANIZATION_BLOCK "OB86"   // OB86, LAD, RackStationFailure
{ S7_Optimized_Access := 'TRUE' }
VERSION : 0.1
   VAR_INPUT
      LADDR : Hw_Device;   // Hardware identifier
      Event_Class : Byte;   // Event class
      Fault_ID : Byte;   // Fault identifier
   END_VAR
BEGIN
END_ORGANIZATION_BLOCK

ORGANIZATION_BLOCK "OB100"   // OB100, LAD, Startup
TITLE = "Complete Restart"
{ S7_Optimized_Access := 'TRUE' }
VERSION : 0.1
   VAR_INPUT
      LostRetentive : Bool;   // True if retentive data are lost
      LostRTC : Bool;   // True if date and time are lost
   END_VAR
BEGIN
END_ORGANIZATION_BLOCK

(* ===== HMI "HMI_RT_2" =====
system functions are stored by id; their names below are inferred from use
connection "boiler_conection_s71200": ETHERNET, S7_1200_OMS
connection "Local_boiler_plc_hmi": ETHERNET, S7_1200_OMS

HMI tags "Default tag table"
   "ALARM_1" : Word AT %MW14, 1 s
   "ALARM_2" : Word AT %MW16, 1 s
   "ANALOG_DISPLAY.CO2_LEVEL" : Real AT %DB102.DBD52, 1 s
   "ANALOG_DISPLAY.FLUE_GAS_TEMP" : Real AT %DB102.DBD60, 1 s
   "ANALOG_DISPLAY.FP1_SPEED" : Real AT %DB102.DBD20, 1 s
   "ANALOG_DISPLAY.FP2_SPEED" : Real AT %DB102.DBD24, 1 s
   "ANALOG_DISPLAY.ID_SPEED" : Real AT %DB102.DBD28, 1 s
   "ANALOG_DISPLAY.LH_BURNBACK_TEMP" : Real AT %DB102.DBD64, 1 s
   "ANALOG_DISPLAY.LH_FRONT_UND_POS" : Real AT %DB102.DBD72, 1 s
   "ANALOG_DISPLAY.LH_REAR_UND_POS" : Real AT %DB102.DBD80, 1 s
   "ANALOG_DISPLAY.LH_TOTAL_COAL" : Real AT %DB102.DBD100, 1 s
   "ANALOG_DISPLAY.LHFD_SPEED" : Real AT %DB102.DBD32, 1 s
   "ANALOG_DISPLAY.LHSTOKER_SPEED" : Real AT %DB102.DBD40, 1 s
   "ANALOG_DISPLAY.O2_LEVEL" : Real AT %DB102.DBD48, 1 s
   "ANALOG_DISPLAY.PUMP_PRESSURE" : Real AT %DB102.DBD8, 1 s
   "ANALOG_DISPLAY.RH_BURNBACK_TEMP" : Real AT %DB102.DBD68, 1 s
   "ANALOG_DISPLAY.RH_FRONT_UND_POS" : Real AT %DB102.DBD76, 1 s
   "ANALOG_DISPLAY.RH_REAR_UND_POS" : Real AT %DB102.DBD84, 1 s
   "ANALOG_DISPLAY.RH_TOTAL_COAL" : Real AT %DB102.DBD104, 1 s
   "ANALOG_DISPLAY.RHFD_SPEED" : Real AT %DB102.DBD36, 1 s
   "ANALOG_DISPLAY.RHSTOKER_SPEED" : Real AT %DB102.DBD44, 1 s
   "ANALOG_DISPLAY.STEAM_PRESSURE" : Real AT %DB102.DBD4, 1 s
   "ANALOG_DISPLAY.TOTAL_WATER" : Real AT %DB102.DBD96, 1 s
   "ANALOG_DISPLAY.WATER_FLOWRATE" : Real AT %DB102.DBD12, 1 s
   "ANALOG_DISPLAY.WATER_LEVEL" : Real AT %DB102.DBD0, 1 s
   "ANALOG_DISPLAY.WATER_TEMP" : Real AT %DB102.DBD56, 1 s
   "ANALOG_DISPLAY.WATER_TEMP_ECO" : Real AT %DB102.DBD108, 1 s
   "DATA_PARAMETER.DELAY_TIME_LH_BUCKET" : Time AT %DB106.DBD270, 1 s
   "DATA_PARAMETER.DELAY_TIME_RH_BUCKET" : Time AT %DB106.DBD274, 1 s
   "DATA_PARAMETER.GAIN_FD" : Real AT %DB201.DBD36, 1 s
   "DATA_PARAMETER.GAIN_PUMPS" : Real AT %DB106.DBD322, 1 s
   "DATA_PARAMETER.HAND_REFF_FP" : Real AT %DB106.DBD16, 1 s
   "DATA_PARAMETER.HAND_REFF_LHFRONT_UND" : Real AT %DB106.DBD108, 1 s
   "DATA_PARAMETER.HAND_REFF_LHREAR_UND" : Real AT %DB106.DBD116, 1 s
   "DATA_PARAMETER.HAND_REFF_RHFRONT_UND" : Real AT %DB106.DBD112, 1 s
   "DATA_PARAMETER.HAND_REFF_RHREAR_UND" : Real AT %DB106.DBD120, 1 s
   "DATA_PARAMETER.HL_HIGH_LIMIT" : Real AT %DB106.DBD36, 1 s
   "DATA_PARAMETER.HL_LOW_LIMIT" : Real AT %DB106.DBD28, 1 s
   "DATA_PARAMETER.HSP_ID_FAN" : Real AT %DB106.DBD72, 1 s
   "DATA_PARAMETER.HSP_LH_STOKER" : Real AT %DB106.DBD92, 1 s
   "DATA_PARAMETER.HSP_LHFD_FAN" : Real AT %DB106.DBD84, 1 s
   "DATA_PARAMETER.HSP_RH_STOKER" : Real AT %DB106.DBD242, 1 s
   "DATA_PARAMETER.HSP_RHFD_FAN" : Real AT %DB106.DBD210, 1 s
   "DATA_PARAMETER.LH_COAL_HEIGHT" : Real AT %DB106.DBD156, 1 s
   "DATA_PARAMETER.LH_DENSITY" : Real AT %DB106.DBD164, 1 s
   "DATA_PARAMETER.LH_OFFSET" : DInt AT %DB106.DBD100, 1 s
   "DATA_PARAMETER.LL_HIGH_LIMIT" : Real AT %DB106.DBD32, 1 s
   "DATA_PARAMETER.LL_LOW_LIMIT" : Real AT %DB106.DBD24, 1 s
   "DATA_PARAMETER.LSP_ID_FAN" : Real AT %DB106.DBD68, 1 s
   "DATA_PARAMETER.LSP_LH_STOKER" : Real AT %DB106.DBD88, 1 s
   "DATA_PARAMETER.LSP_LHFD_FAN" : Real AT %DB106.DBD80, 1 s
   "DATA_PARAMETER.LSP_PUMPS" : Real AT %DB106.DBD338, 1 s
   "DATA_PARAMETER.LSP_RH_STOKER" : Real AT %DB106.DBD238, 1 s
   "DATA_PARAMETER.LSP_RHFD_FAN" : Real AT %DB106.DBD206, 1 s
   "DATA_PARAMETER.MAX_FLOWRATE" : Real AT %DB106.DBD20, 1 s
   "DATA_PARAMETER.MAX_FRONT_LHUND" : Real AT %DB106.DBD124, 1 s
   "DATA_PARAMETER.MAX_FRONT_RHUND" : Real AT %DB106.DBD132, 1 s
   "DATA_PARAMETER.MAX_PERC_O2" : Real AT %DB201.DBD24, 1 s
   "DATA_PARAMETER.MIN_FRONT_LHUND" : Real AT %DB106.DBD128, 1 s
   "DATA_PARAMETER.MIN_FRONT_RHUND" : Real AT %DB106.DBD136, 1 s
   "DATA_PARAMETER.OFF_PULSE_BLOWDOWN" : Time AT %DB106.DBD176, 1 s
   "DATA_PARAMETER.OFF_TIME_BLOWDOWN" : Int AT %DB106.DBW346, 1 s
   "DATA_PARAMETER.ON_DELAY_FD_DECREASE" : Time AT %DB106.DBD294, 1 s
   "DATA_PARAMETER.ON_PULSE_BLOWDOWN" : Time AT %DB106.DBD180, 1 s
   "DATA_PARAMETER.PERIODE" : Int AT %DB106.DBW184, 1 s
   "DATA_PARAMETER.RH_COAL_HEIGHT" : Real AT %DB106.DBD160, 1 s
   "DATA_PARAMETER.RH_DENSITY" : Real AT %DB106.DBD168, 1 s
   "DATA_PARAMETER.RH_OFFSET" : DInt AT %DB106.DBD104, 1 s
   "DATA_PARAMETER.SP_ECO" : Real AT %DB106.DBD202, 1 s
   "DATA_PARAMETER.SP_FD" : Real AT %DB106.DBD4, 1 s
   "DATA_PARAMETER.SP_O2" : Real AT %DB106.DBD306, 1 s
   "DATA_PARAMETER.SP_STOKER" : Real AT %DB106.DBD8, 1 s
   "DATA_PARAMETER.SP_WATER_LEVEL" : Real AT %DB106.DBD0, 1 s
   "DATA_PARAMETER.TD_FD" : Real AT %DB201.DBD44, 1 s
   "DATA_PARAMETER.TD_PUMPS" : Real AT %DB106.DBD330, 1 s
   "DATA_PARAMETER.TI_FD" : Real AT %DB201.DBD40, 1 s
   "DATA_PARAMETER.TI_PUMPS" : Real AT %DB106.DBD326, 1 s
   "DATA_STATUS.ASH_CONV_STATUS" : Int AT %DB154.DBW22, 1 s
   "DATA_STATUS.COAL_CONV1_STATUS" : Int AT %DB154.DBW40, 1 s
   "DATA_STATUS.COAL_CONV2_STATUS" : Int AT %DB154.DBW42, 1 s
   "DATA_STATUS.FP1_STATUS" : Int AT %DB154.DBW0, 1 s
   "DATA_STATUS.FP2_STATUS" : Int AT %DB154.DBW2, 1 s
   "DATA_STATUS.IDFAN_STATUS" : Int AT %DB154.DBW4, 1 s
   "DATA_STATUS.LH_STOKER_STATUS" : Int AT %DB154.DBW10, 1 s
   "DATA_STATUS.LH_SWING_STATUS" : Int AT %DB154.DBW14, 1 s
   "DATA_STATUS.LHFD_FAN_STATUS" : Int AT %DB154.DBW6, 1 s
   "DATA_STATUS.RAV1_STATUS" : Int AT %DB154.DBW18, 1 s
   "DATA_STATUS.RAV2_STATUS" : Int AT %DB154.DBW20, 1 s
   "DATA_STATUS.RH_STOKER_STATUS" : Int AT %DB154.DBW12, 1 s
   "DATA_STATUS.RH_SWING_STATUS" : Int AT %DB154.DBW16, 1 s
   "DATA_STATUS.RHFD_FAN_STATUS" : Int AT %DB154.DBW8, 1 s
   "DATA_STATUS.WET_SCRUBBER_PUMP_STATUS" : Int AT %DB154.DBW32, 1 s
   "DATA_SWITCH.AUTO_ECO" : Bool AT %DB101.DBX8.7, 1 s
   "DATA_SWITCH.AUTO_FP" : Bool AT %DB101.DBX0.0, 1 s
   "DATA_SWITCH.AUTO_ID" : Bool AT %DB101.DBX1.2, 1 s
   "DATA_SWITCH.AUTO_LH_BUCKET" : Bool AT %DB101.DBX7.0, 1 s
   "DATA_SWITCH.AUTO_LHFD" : Bool AT %DB101.DBX1.3, 1 s
   "DATA_SWITCH.AUTO_LHFRONT_UND_SW" : Bool AT %DB101.DBX5.1, 1 s
   "DATA_SWITCH.AUTO_LHSTOKER" : Bool AT %DB101.DBX1.4, 1 s
   "DATA_SWITCH.AUTO_LHSWING" : Bool AT %DB101.DBX1.6, 1 s
   "DATA_SWITCH.AUTO_RH_BUCKET" : Bool AT %DB101.DBX7.1, 1 s
   "DATA_SWITCH.AUTO_RHFD" : Bool AT %DB101.DBX6.3, 1 s
   "DATA_SWITCH.AUTO_RHFRONT_UND_SW" : Bool AT %DB101.DBX5.2, 1 s
   "DATA_SWITCH.AUTO_RHSTOKER" : Bool AT %DB101.DBX1.5, 1 s
   "DATA_SWITCH.AUTO_RHSWING" : Bool AT %DB101.DBX1.7, 1 s
   "DATA_SWITCH.COAL_CONV1_SW_HMI" : Bool AT %DB101.DBX7.2, 1 s
   "DATA_SWITCH.COAL_CONV2_SW_HMI" : Bool AT %DB101.DBX7.6, 1 s
   "DATA_SWITCH.HAND_CLOSE_ECO" : Bool AT %DB101.DBX9.1, 1 s
   "DATA_SWITCH.HAND_LH_FRONT_UND_CLOSE" : Bool AT %DB101.DBX10.0, 1 s
   "DATA_SWITCH.HAND_LH_FRONT_UND_OPEN" : Bool AT %DB101.DBX9.7, 1 s
   "DATA_SWITCH.HAND_LH_REAR_UND_CLOSE" : Bool AT %DB101.DBX10.5, 1 s
   "DATA_SWITCH.HAND_LH_REAR_UND_OPEN" : Bool AT %DB101.DBX10.4, 1 s
   "DATA_SWITCH.HAND_OPEN_ECO" : Bool AT %DB101.DBX9.0, 1 s
   "DATA_SWITCH.HAND_RH_FRONT_UND_CLOSE" : Bool AT %DB101.DBX10.2, 1 s
   "DATA_SWITCH.HAND_RH_FRONT_UND_OPEN" : Bool AT %DB101.DBX10.1, 1 s
   "DATA_SWITCH.HAND_RH_REAR_UND_CLOSE" : Bool AT %DB101.DBX10.7, 1 s
   "DATA_SWITCH.HAND_RH_REAR_UND_OPEN" : Bool AT %DB101.DBX10.6, 1 s
   "DATA_SWITCH.HAND_SPEED_DOWN_ID" : Bool AT %DB101.DBX3.2, 1 s
   "DATA_SWITCH.HAND_SPEED_DOWN_LHFD" : Bool AT %DB101.DBX3.4, 1 s
   "DATA_SWITCH.HAND_SPEED_DOWN_LHSTOKER" : Bool AT %DB101.DBX4.0, 1 s
   "DATA_SWITCH.HAND_SPEED_DOWN_RHFD" : Bool AT %DB101.DBX3.6, 1 s
   "DATA_SWITCH.HAND_SPEED_DOWN_RHSTOKER" : Bool AT %DB101.DBX4.2, 1 s
   "DATA_SWITCH.HAND_SPEED_UP_ID" : Bool AT %DB101.DBX3.1, 1 s
   "DATA_SWITCH.HAND_SPEED_UP_LHFD" : Bool AT %DB101.DBX3.3, 1 s
   "DATA_SWITCH.HAND_SPEED_UP_LHSTOKER" : Bool AT %DB101.DBX3.7, 1 s
   "DATA_SWITCH.HAND_SPEED_UP_RHFD" : Bool AT %DB101.DBX3.5, 1 s
   "DATA_SWITCH.HAND_SPEED_UP_RHSTOKER" : Bool AT %DB101.DBX4.1, 1 s
   "DATA_SWITCH.LH_HAND_BUCKET_DOWN" : Bool AT %DB101.DBX6.6, 1 s
   "DATA_SWITCH.LH_HAND_BUCKET_UP" : Bool AT %DB101.DBX6.5, 1 s
   "DATA_SWITCH.O2_CONTROL_ENABLE_SW" : Bool AT %DB101.DBX10.3, 1 s
   "DATA_SWITCH.RH_HAND_BUCKET_DOWN" : Bool AT %DB101.DBX6.7, 1 s
   "DATA_SWITCH.RH_HAND_BUCKET_UP" : Bool AT %DB101.DBX8.6, 1 s
   "DATA_SWITCH.SW_ASH_CONV" : Bool AT %DB101.DBX0.7, 1 s
   "DATA_SWITCH.SW_LHSTOKER" : Bool AT %DB101.DBX0.5, 1 s
   "DATA_SWITCH.SW_LHSWING" : Bool AT %DB101.DBX1.0, 1 s
   "DATA_SWITCH.SW_RHSTOKER" : Bool AT %DB101.DBX0.6, 1 s
   "DATA_SWITCH.SW_RHSWING" : Bool AT %DB101.DBX1.1, 1 s
   "DATA_SWITCH.SW_WETSCRUBBER" : Bool AT %DB101.DBX3.0, 1 s
   "FP_PRESSURE.SP_H" : Real AT %DB108.DBD20, 1 s   // Alarm Setpoint: High
   "LH_BURNBACK_TEMP.SP_H" : Real = PLC DB129_LH_BURNBACK_TEMP.IN7 AT %DB129.DBD20, 1 s   // Alarm Setpoint: High
   "LHFD_SCALING.Value" : Real = PLC DB173_LHFD_SCALING.Out13 AT %DB173.DBD30, 1 s   // Scaled engineering value
   "PID_STOKER.GAIN" : Real AT %DB201.DBD4, 1 s   // proportional gain
   "PID_STOKER.TD" : Real AT %DB201.DBD12, 1 s   // derivative time
   "PID_STOKER.TI" : Real AT %DB201.DBD8, 1 s   // reset time
   "RH_BURNBACK_TEMP.SP_H" : Real = PLC DB130_RH_BURNBACK_TEMP.IN7 AT %DB130.DBD20, 1 s   // Alarm Setpoint: High
   "RH_FD_SCALING.Value" : Real = PLC DB176_RH_FD_SCALING.Out13 AT %DB176.DBD30, 1 s   // Scaled engineering value
   "STEAM_PRESS.SP_H" : Real = PLC DB109_STEAM_PRESS.IN7 AT %DB109.DBD20, 1 s   // Alarm Setpoint: High
   "STEAM_PRESS.SP_L" : Real = PLC DB109_STEAM_PRESS.IN6 AT %DB109.DBD16, 1 s   // Alarm Setpoint: Low
   "WORK_BIT.ECO_CLOSE" : Bool AT %DB100.DBX16.2, 1 s
   "WORK_BIT.ECO_OPEN" : Bool AT %DB100.DBX16.1, 1 s
   "WORK_BIT.LH_FRONT_UND_CLOSE" : Bool AT %DB100.DBX19.7, 1 s
   "WORK_BIT.LH_FRONT_UND_OPEN" : Bool AT %DB100.DBX19.6, 1 s
   "WORK_BIT.LH_REAR_UND_CLOSED" : Bool AT %DB100.DBX20.3, 1 s
   "WORK_BIT.LH_REAR_UND_OPEN" : Bool AT %DB100.DBX20.2, 1 s
   "WORK_BIT.LH_SINGLE_BUCKET_DOWN" : Bool AT %DB100.DBX19.3, 1 s
   "WORK_BIT.LH_SINGLE_BUCKET_UP" : Bool AT %DB100.DBX19.2, 1 s
   "WORK_BIT.MPA_26" : Bool AT %DB100.DBX2.3, 1 s
   "WORK_BIT.RH_FRONT_UND_CLOSE" : Bool AT %DB100.DBX20.1, 1 s
   "WORK_BIT.RH_FRONT_UND_OPEN" : Bool AT %DB100.DBX20.0, 1 s
   "WORK_BIT.RH_REAR_UND_CLOSED" : Bool AT %DB100.DBX20.5, 1 s
   "WORK_BIT.RH_REAR_UND_OPEN" : Bool AT %DB100.DBX20.4, 1 s
   "WORK_BIT.RH_SINGLE_BUCKET_DOWN" : Bool AT %DB100.DBX19.5, 1 s
   "WORK_BIT.RH_SINGLE_BUCKET_UP" : Bool AT %DB100.DBX19.4, 1 s
   "WTR_LEVEL_SCALING.SP_H" : Real = PLC DB104_WTR_LEVEL_SCALING.IN7 AT %DB104.DBD20, 1 s   // Alarm Setpoint: High
   "WTR_LEVEL_SCALING.SP_L" : Real = PLC DB104_WTR_LEVEL_SCALING.IN6 AT %DB104.DBD16, 1 s   // Alarm Setpoint: Low
   "SP_FD_FAN" : Real AT %DB201.DBD32, 1 s
   "PB_BLOWDOWN" : Bool AT %DB101.DBX11.3, 1 s
   "Hand/Auto_Blowdown" : Bool AT %DB101.DBX11.2, 1 s
   "PUMP_SPEED_UP" : Bool, internal
   "PUMP_SPEED_DOWN" : Bool, internal
   "PID_STROKER_SETPOINT" : Real AT %DB201.DBD0, 1 s
   "Change_Date_1" : Bool, internal
   "Change_Time_1" : Bool, internal
   "Out_PID_FD" : Real AT %DB106.DBD76, 1 s
   "Out_PID_PUMP" : Real AT %DB106.DBD334, 1 s
   "Out_PID_STOKER" : Real AT %DB106.DBD96, 1 s
   "Set_Date_Time" : DTL AT %DB1.DBX2.0, 1 s
   "Date_Time_Actual" : DTL AT %DB1.DBX16.0, 1 s
   "Set_DTL" : Bool AT %DB1.DBX50.0, 1 s
   "LH_BURN_BACK_OFFSET" : Real AT %DB9.DBD4, 1 s
   "RH_BURN_BACK_OFFSET" : Real AT %DB9.DBD12, 1 s
   "Clock_1s" : Bool AT %M10.5, 1 s

HMI tags "AI Min Max"
   "DB_Scalling_Pressurre_Steam_Min" : Real = PLC DB_Scalling.Pressurre_Steam_Min AT %DB21.DBD0, 1 s
   "DB_Scalling_Pressure_Steam_Max" : Real = PLC DB_Scalling.Pressure_Steam_Max AT %DB21.DBD4, 1 s
   "DB_Scalling_Pressure_Pump_Min" : Real = PLC DB_Scalling.Pressure_Pump_Min AT %DB21.DBD8, 1 s
   "DB_Scalling_Pressure_Pump_Max" : Real = PLC DB_Scalling.Pressure_Pump_Max AT %DB21.DBD12, 1 s
   "DB_Scalling_Water_Flowrate_Min" : Real = PLC DB_Scalling.Water_Flowrate_Min AT %DB21.DBD16, 1 s
   "DB_Scalling_Water_Flowrate_Max" : Real = PLC DB_Scalling.Water_Flowrate_Max AT %DB21.DBD20, 1 s
   "DB_Scalling_Feed_Pump_1_Min" : Real = PLC DB_Scalling.Feed_Pump_1_Min AT %DB21.DBD24, 1 s
   "DB_Scalling_Feed_Pump_1_Max" : Real = PLC DB_Scalling.Feed_Pump_1_Max AT %DB21.DBD28, 1 s
   "DB_Scalling_Feed_Pump_2_Min" : Real = PLC DB_Scalling.Feed_Pump_2_Min AT %DB21.DBD32, 1 s
   "DB_Scalling_Feed_Pump_2_Max" : Real = PLC DB_Scalling.Feed_Pump_2_Max AT %DB21.DBD36, 1 s
   "DB_Scalling_ID_Fan_Min" : Real = PLC DB_Scalling.ID_Fan_Min AT %DB21.DBD40, 1 s
   "DB_Scalling_ID_Fan_Max" : Real = PLC DB_Scalling.ID_Fan_Max AT %DB21.DBD44, 1 s
   "DB_Scalling_LH_FD_Fan_Min" : Real = PLC DB_Scalling.LH_FD_Fan_Min AT %DB21.DBD48, 1 s
   "DB_Scalling_LH_FD_Fan_Max" : Real = PLC DB_Scalling.LH_FD_Fan_Max AT %DB21.DBD52, 1 s
   "DB_Scalling_RH_FD_Fan_Min" : Real = PLC DB_Scalling.RH_FD_Fan_Min AT %DB21.DBD56, 1 s
   "DB_Scalling_RH_FD_Fan_Max" : Real = PLC DB_Scalling.RH_FD_Fan_Max AT %DB21.DBD60, 1 s
   "DB_Scalling_LH_Stoker_Min" : Real = PLC DB_Scalling.LH_Stoker_Min AT %DB21.DBD64, 1 s
   "DB_Scalling_LH_Stoker_Max" : Real = PLC DB_Scalling.LH_Stoker_Max AT %DB21.DBD68, 1 s
   "DB_Scalling_RH_Stoker_Min" : Real = PLC DB_Scalling.RH_Stoker_Min AT %DB21.DBD72, 1 s
   "DB_Scalling_RH_Stoker_Max" : Real = PLC DB_Scalling.RH_Stoker_Max AT %DB21.DBD76, 1 s
   "DB_Scalling_NRGT(Water_Level)_Min" : Real = PLC DB_Scalling.NRGT(Water_Level)_Min AT %DB21.DBD80, 1 s
   "DB_Scalling_NRGT(Water_Level)_Max" : Real = PLC DB_Scalling.NRGT(Water_Level)_Max AT %DB21.DBD84, 1 s
   "DB_Scalling_O2_Probe_Min" : Real = PLC DB_Scalling.O2_Probe_Min AT %DB21.DBD88, 1 s
   "DB_Scalling_O2_Probe_Max" : Real = PLC DB_Scalling.O2_Probe_Max AT %DB21.DBD92, 1 s
   "DB_Scalling_Water_Temp_Min" : Real = PLC DB_Scalling.Water_Temp_Min AT %DB21.DBD96, 1 s
   "DB_Scalling_Water_Temp_Max" : Real = PLC DB_Scalling.Water_Temp_Max AT %DB21.DBD100, 1 s
   "DB_Scalling_Flue_Min" : Real = PLC DB_Scalling.Flue_Min AT %DB21.DBD104, 1 s
   "DB_Scalling_Flue_Max" : Real = PLC DB_Scalling.Flue_Max AT %DB21.DBD108, 1 s
   "DB_Scalling_LH_Thermocouple_Min" : Real = PLC DB_Scalling.LH_Thermocouple_Min AT %DB21.DBD112, 1 s
   "DB_Scalling_LH_Thermocouple_Max" : Real = PLC DB_Scalling.LH_Thermocouple_Max AT %DB21.DBD116, 1 s
   "DB_Scalling_RH_Thermocouple_Min" : Real = PLC DB_Scalling.RH_Thermocouple_Min AT %DB21.DBD120, 1 s
   "DB_Scalling_RH_Thermocouple_Max" : Real = PLC DB_Scalling.RH_Thermocouple_MAX AT %DB21.DBD124, 1 s
   "DB_Scalling_LH_Front_Undergrate_Min" : Real = PLC DB_Scalling.LH_Front_Undergrate_Min AT %DB21.DBD128, 1 s
   "DB_Scalling_LH_Front_Undergrate_Max" : Real = PLC DB_Scalling.LH_Front_Undergrate_Max AT %DB21.DBD132, 1 s
   "DB_Scalling_RH_Front_Undergrate_Min" : Real = PLC DB_Scalling.RH_Front_Undergrate_Min AT %DB21.DBD136, 1 s
   "DB_Scalling_RH_Front_Undergrate_Max" : Real = PLC DB_Scalling.RH_Front_Undergrate_Max AT %DB21.DBD140, 1 s
   "DB_Scalling_LH_Rear_Undergrate_Min" : Real = PLC DB_Scalling.LH_Rear_Undergrate_Min AT %DB21.DBD144, 1 s
   "DB_Scalling_LH_Rear_Undergrate_Max" : Real = PLC DB_Scalling.LH_Rear_Undergrate_Max AT %DB21.DBD148, 1 s
   "DB_Scalling_RH_Rear_Undergrate_Min" : Real = PLC DB_Scalling.RH_Rear_Undergrate_Min AT %DB21.DBD152, 1 s
   "DB_Scalling_RH_Rear_Undergrate_Max" : Real = PLC DB_Scalling.RH_Rear_Undergrate_Max AT %DB21.DBD156, 1 s
   "DB_Scalling_Analog_LH_Front_Min" : Real = PLC DB_Scalling.Analog_LH_Front_Min AT %DB21.DBD160, 1 s
   "DB_Scalling_Analog_LH_Front_Max" : Real = PLC DB_Scalling.Analog_LH_Front_Max AT %DB21.DBD164, 1 s
   "DB_Scalling_Analog_RH_Front_Min" : Real = PLC DB_Scalling.Analog_RH_Front_Min AT %DB21.DBD168, 1 s
   "DB_Scalling_Analog_RH_Front_Max" : Real = PLC DB_Scalling.Analog_RH_Front_Max AT %DB21.DBD172, 1 s
   "DB_Scalling_Analog_LH_Rear_Min" : Real = PLC DB_Scalling.Analog_LH_Rear_Min AT %DB21.DBD176, 1 s
   "DB_Scalling_Analog_LH_Rear_Max" : Real = PLC DB_Scalling.Analog_LH_Rear_Max AT %DB21.DBD180, 1 s
   "DB_Scalling_Analog_RH_Rear_Min" : Real = PLC DB_Scalling.Analog_RH_Rear_Min AT %DB21.DBD184, 1 s
   "DB_Scalling_Analog_RH_Rear_Max" : Real = PLC DB_Scalling.Analog_RH_Rear_Max AT %DB21.DBD188, 1 s
   "DB103_ANALOG_INPUT_STAT15_Poti LH Front Undgrt" : Int = PLC DB103_ANALOG_INPUT."STAT15_Poti LH Front Undgrt" AT %DB103.DBW30, 1 s
   "DB103_ANALOG_INPUT_STAT16_Poti RH Front Undgrt" : Int = PLC DB103_ANALOG_INPUT."STAT16_Poti RH Front Undgrt" AT %DB103.DBW32, 1 s
   "DB103_ANALOG_INPUT_STAT17_Poti LH Rear Undgrt" : Int = PLC DB103_ANALOG_INPUT."STAT17_Poti LH Rear Undgrt" AT %DB103.DBW34, 1 s
   "DB103_ANALOG_INPUT_STAT18_Poti RH Rear Undgrt" : Int = PLC DB103_ANALOG_INPUT."STAT18_Poti RH Rear Undgrt" AT %DB103.DBW36, 1 s

discrete alarms
   25: 'WET SCRUBBER FAULT', class Warnings, trigger "ALARM_2" bit 8
   24: 'EMERGENCY STOP', class Errors, trigger "ALARM_2" bit 7
   27: 'WATER FLOWRATE FAULT', class Warnings, trigger "ALARM_2" bit 10
   20: 'LOCKOUT', class Errors, trigger "ALARM_2" bit 3
   28: 'LH SINGLE BUCKET FAULT', class Warnings, trigger "ALARM_2" bit 11
   18: 'LH BURNBACK FAULT', class Warnings, trigger "ALARM_2" bit 1
   22: 'STEAM PRESSURE TOO LOW', class Warnings, trigger "ALARM_2" bit 5
   17: 'RH SHEARPIN FAULT', class Warnings, trigger "ALARM_2" bit 0
   30: 'FP DRY RUN PROTECTION', class Warnings, trigger "ALARM_2" bit 13
   21: 'COAL HOPPER LOW LEVEL', class Warnings, trigger "ALARM_2" bit 4
   26: 'PUMP PRESSURE LOW', class Warnings, trigger "ALARM_2" bit 9
   19: 'RH BURNBACK FAULT', class Warnings, trigger "ALARM_2" bit 2
   11: 'LH SWING CHUTE FAULT', class Warnings, trigger "ALARM_1" bit 10
   5: 'FEED PUMP 2 FAULT', class Warnings, trigger "ALARM_1" bit 4
   7: 'LH FD FAN FAULT', class Warnings, trigger "ALARM_1" bit 6
   9: 'LH STOKER FAULT', class Warnings, trigger "ALARM_1" bit 8
   6: 'ID FAN FAULT', class Errors, trigger "ALARM_1" bit 5
   3: 'HIGH WATER', class Warnings, trigger "ALARM_1" bit 2
   10: 'RH STOKER FAULT', class Warnings, trigger "ALARM_1" bit 9
   4: 'FEED PUMP 1 FAULT', class Warnings, trigger "ALARM_1" bit 3
   1: 'LOW WATER PREWARNING', class Warnings, trigger "ALARM_1" bit 0
   14: 'RAV2 FAULT', class Warnings, trigger "ALARM_1" bit 13
   8: 'RH FD FAN FAULT', class Warnings, trigger "ALARM_1" bit 7
   12: 'RH SWING CHUTE FAULT', class Warnings, trigger "ALARM_1" bit 11
   16: 'LH SHEARPIN FAULT', class Warnings, trigger "ALARM_1" bit 15
   15: 'ASH CONVEYOR FAULT', class Warnings, trigger "ALARM_1" bit 14
   13: 'RAV1 FAULT', class Warnings, trigger "ALARM_1" bit 12
   23: 'STEAM PRESSURE TOO HIGH', class Warnings, trigger "ALARM_2" bit 6
   29: 'RH SINGLE BUCKET FAULT', class Warnings, trigger "ALARM_2" bit 12
   2: 'LOW WATER', class Errors, trigger "ALARM_1" bit 1

analog alarms
   13: 'The value is above upper limit', class Warnings, trigger "DATA_PARAMETER.SP_WATER_LEVEL"
   7: 'The value is above upper limit', class Warnings, trigger "DATA_PARAMETER.HAND_REFF_LHFRONT_UND"
   4: 'The value is below lower limit', class Warnings, trigger "DATA_PARAMETER.HAND_REFF_LHREAR_UND"
   3: 'The value is above upper limit', class Warnings, trigger "DATA_PARAMETER.HAND_REFF_LHREAR_UND"
   10: 'The value is below lower limit', class Warnings, trigger "DATA_PARAMETER.HAND_REFF_RHFRONT_UND"
   9: 'The value is above upper limit', class Warnings, trigger "DATA_PARAMETER.HAND_REFF_RHFRONT_UND"
   6: 'The value is below lower limit', class Warnings, trigger "DATA_PARAMETER.HAND_REFF_RHREAR_UND"
   5: 'The value is above upper limit', class Warnings, trigger "DATA_PARAMETER.HAND_REFF_RHREAR_UND"
   8: 'The value is below lower limit', class Warnings, trigger "DATA_PARAMETER.HAND_REFF_LHFRONT_UND"
   11: 'The value is above upper limit', class Warnings, trigger "DATA_PARAMETER.LH_OFFSET"
   12: 'The value is below lower limit', class Warnings, trigger "DATA_PARAMETER.LH_OFFSET"
   1: 'The value is above upper limit', class Warnings, trigger "DATA_PARAMETER.SP_FD"
   2: 'The value is below lower limit', class Warnings, trigger "DATA_PARAMETER.SP_FD"

screen "Stoker" 1280x800, template "Template_All"
   TextField "Text field_1" at 312,216 size 170x43; Text 'LH STOKER'
   TextField "Text field_2" at 838,216 size 174x43; Text 'RH STOKER'
   TextField "Text field_3" at 408,116 size 419x44; Text 'CHAIN GRATE STOKER'
   Button "Button_1" at 0,730 size 98x68; TextOff 'Text'; PictureOn "Home_1"; PictureOff "Home_1"
      on Click: ActivateScreen("Home Screen", 0)
   Button "Button_2" at 98,730 size 100x68; TextOn 'Pumps'; TextOff 'Pumps'
      on Click: ActivateScreen("Feed Pump", 0)
   Button "Button_3" at 198,730 size 90x68; TextOn 'Fans'; TextOff 'Fans'
      on Click: ActivateScreen("ID FD Fan", 0)
   Button "Button_4" at 288,730 size 100x68; TextOn 'Stoker'; TextOff 'Stoker'
      on Click: ActivateScreen("Stoker", 0)
   Button "Button_6" at 516,730 size 89x68; TextOff 'Setup'
      on Click: ActivateScreen("Setup", 0)
   Button "Button_11" at 1164,730 size 114x68; TextOff 'Trends'
      on Click: ActivateScreen("Trend Steam", 0)
   Button "Button_5" at 387,730 size 129x68; TextOff 'Coal Handling'
      on Click: ActivateScreen("Coal Handling", 0)
   Button "Button_7" at 604,730 size 210x68; TextOff 'Coal & Blowdown Setup'
      on Click: ActivateScreen("Coal Setup", 0)
   Button "Button_8" at 814,730 size 140x68; TextOff 'Front/Rear Undergrate'
      on Click: ActivateScreen("Front Undergrate Damper", 0)
   Button "Button_20" at 954,730 size 100x68; TextOff 'Alarm Setup'
      on Click: ActivateScreen("Alarm Setup", 0)
   Button "Button_21" at 1054,730 size 110x68; TextOff 'Alarm History'
      on Click: ActivateScreen("Alarm History", 0)
   Bar "Bar_3" at 162,280 size 106x414; MinimumValue 0; MaximumValue 60
      ProcessValue <- "ANALOG_DISPLAY.LHSTOKER_SPEED"
   Bar "Bar_4" at 708,280 size 106x414; MinimumValue 0; MaximumValue 60
      ProcessValue <- "ANALOG_DISPLAY.RHSTOKER_SPEED"
   Switch "Switch_2" at 363,362 size 224x80; TextOn 'AUTO'; CaptionText 'Switch'; TextOff 'HAND'
      ProcessValue <- "DATA_SWITCH.AUTO_LHSTOKER"
      Appearance <- "DATA_SWITCH.AUTO_LHSTOKER"
   Button "Button_10" at 363,444 size 224x80; TextOff 'SPEED UP'
      on Press: function_b14e0dd5("DATA_SWITCH.HAND_SPEED_UP_LHSTOKER", 0)
      Appearance <- "DATA_SWITCH.HAND_SPEED_UP_LHSTOKER"
   Button "Button_9" at 363,526 size 224x80; TextOff 'SPEED DOWN'
      on Press: function_b14e0dd5("DATA_SWITCH.HAND_SPEED_DOWN_LHSTOKER", 0)
      Appearance <- "DATA_SWITCH.HAND_SPEED_DOWN_LHSTOKER"
   IOField "IO Field_2" at 363,608 size 224x80; FormatPattern 99.9
      ProcessValue <- "ANALOG_DISPLAY.LHSTOKER_SPEED"
   Switch "Switch_3" at 363,280 size 224x80; TextOn 'RUN'; CaptionText 'Switch'; TextOff 'STOP'
      ProcessValue <- "DATA_SWITCH.SW_LHSTOKER"
      Appearance <- "DATA_STATUS.LH_STOKER_STATUS"
   Switch "Switch_4" at 890,362 size 224x80; TextOn 'AUTO'; CaptionText 'Switch'; TextOff 'HAND'
      ProcessValue <- "DATA_SWITCH.AUTO_RHSTOKER"
      Appearance <- "DATA_SWITCH.AUTO_RHSTOKER"
   Button "Button_22" at 890,444 size 224x80; TextOff 'SPEED UP'
      on Press: function_b14e0dd5("DATA_SWITCH.HAND_SPEED_UP_RHSTOKER", 0)
      Appearance <- "DATA_SWITCH.HAND_SPEED_UP_RHSTOKER"
   Button "Button_23" at 890,526 size 224x80; TextOff 'SPEED DOWN'
      on Press: function_b14e0dd5("DATA_SWITCH.HAND_SPEED_DOWN_RHSTOKER", 0)
      Appearance <- "DATA_SWITCH.HAND_SPEED_DOWN_RHSTOKER"
   IOField "IO Field_3" at 890,608 size 224x80; FormatPattern 99.9
      ProcessValue <- "ANALOG_DISPLAY.RHSTOKER_SPEED"
   Switch "Switch_5" at 890,280 size 224x80; TextOn 'RUN'; CaptionText 'Switch'; TextOff 'STOP'
      ProcessValue <- "DATA_SWITCH.SW_RHSTOKER"
      Appearance <- "DATA_STATUS.RH_STOKER_STATUS"
   TextField "Text field_4" at 532,631 size 33x34; Text 'Hz'
   TextField "Text field_15" at 1066,631 size 33x34; Text 'Hz'

screen "ID FD Fan" 1280x800, template "Template_All"
   TextField "Text field_3" at 978,251 size 163x43; Text 'RH FD FAN'
   TextField "Text field_15" at 564,251 size 159x43; Text 'LH FD FAN'
   TextField "Text field_16" at 167,249 size 106x43; Text 'ID FAN'
   TextField "Text field_17" at 526,112 size 185x50; Text 'ID-FD FAN'
   Bar "Bar_4" at 45,332 size 92x328; MinimumValue 0; MaximumValue 60
      ProcessValue <- "ANALOG_DISPLAY.ID_SPEED"
   Bar "Bar_2" at 469,332 size 92x328; MinimumValue 0; MaximumValue 60
      ProcessValue <- "ANALOG_DISPLAY.LHFD_SPEED"
   Bar "Bar_3" at 894,332 size 92x328; MinimumValue 0; MaximumValue 60
      ProcessValue <- "ANALOG_DISPLAY.RHFD_SPEED"
   Switch "Switch_1" at 187,328 size 224x80; TextOn 'AUTO'; CaptionText 'Switch'; TextOff 'HAND'
      ProcessValue <- "DATA_SWITCH.AUTO_ID"
      Appearance <- "DATA_SWITCH.AUTO_ID"
   Button "Button_12" at 187,410 size 224x80; TextOff 'SPEED UP'
      on Press: function_b14e0dd5("DATA_SWITCH.HAND_SPEED_UP_ID", 0)
      Appearance <- "DATA_SWITCH.HAND_SPEED_UP_ID"
   Button "Button_13" at 187,492 size 224x80; TextOff 'SPEED DOWN'
      on Press: function_b14e0dd5("DATA_SWITCH.HAND_SPEED_DOWN_ID", 0)
      Appearance <- "DATA_SWITCH.HAND_SPEED_DOWN_ID"
   IOField "IO Field_1" at 187,574 size 224x80; FormatPattern 99.9
      ProcessValue <- "ANALOG_DISPLAY.ID_SPEED"
   TextField "Text field_14" at 364,593 size 35x37; Text 'Hz'
   Switch "Switch_2" at 610,328 size 224x80; TextOn 'AUTO'; CaptionText 'Switch'; TextOff 'HAND'
      ProcessValue <- "DATA_SWITCH.AUTO_LHFD"
      Appearance <- "DATA_SWITCH.AUTO_LHFD"
   Button "Button_14" at 610,410 size 224x80; TextOff 'SPEED UP'
      on Press: function_b14e0dd5("DATA_SWITCH.HAND_SPEED_UP_LHFD", 0)
      Appearance <- "DATA_SWITCH.HAND_SPEED_UP_LHFD"
   Button "Button_15" at 610,492 size 224x80; TextOff 'SPEED DOWN'
      on Press: function_b14e0dd5("DATA_SWITCH.HAND_SPEED_DOWN_LHFD", 0)
      Appearance <- "DATA_SWITCH.HAND_SPEED_DOWN_LHFD"
   IOField "IO Field_2" at 610,574 size 224x80; FormatPattern 99.9
      ProcessValue <- "ANALOG_DISPLAY.LHFD_SPEED"
   TextField "Text field_1" at 787,593 size 35x37; Text 'Hz'
   Switch "Switch_3" at 1033,328 size 224x80; TextOn 'AUTO'; CaptionText 'Switch'; TextOff 'HAND'
      ProcessValue <- "DATA_SWITCH.AUTO_RHFD"
      Appearance <- "DATA_SWITCH.AUTO_RHFD"
   Button "Button_16" at 1033,410 size 224x80; TextOff 'SPEED UP'
      on Release: ResetBit("DATA_SWITCH.HAND_SPEED_UP_RHFD")
      on Press: SetBit("DATA_SWITCH.HAND_SPEED_UP_RHFD")
      Appearance <- "DATA_SWITCH.HAND_SPEED_UP_RHFD"
   Button "Button_17" at 1033,492 size 224x80; TextOff 'SPEED DOWN'
      on Release: ResetBit("DATA_SWITCH.HAND_SPEED_DOWN_RHFD")
      on Press: SetBit("DATA_SWITCH.HAND_SPEED_DOWN_RHFD")
      Appearance <- "DATA_SWITCH.HAND_SPEED_DOWN_RHFD"
   IOField "IO Field_3" at 1033,574 size 224x80; FormatPattern 99.9
      ProcessValue <- "ANALOG_DISPLAY.RHFD_SPEED"
   TextField "Text field_2" at 1210,593 size 35x37; Text 'Hz'
   Switch "Switch_4" at 429,171 size 418x80; TextOn 'O² CONTROL ENABLE'; CaptionText 'Switch'; TextOff 'O² CONTROL DISABLE'
      ProcessValue <- "DATA_SWITCH.O2_CONTROL_ENABLE_SW"
      Appearance <- "DATA_SWITCH.O2_CONTROL_ENABLE_SW"
   Button "Button_1" at 0,730 size 98x68; TextOff 'Text'; PictureOn "Home_1"; PictureOff "Home_1"
      on Click: ActivateScreen("Home Screen", 0)
   Button "Button_2" at 98,730 size 100x68; TextOn 'Pumps'; TextOff 'Pumps'
      on Click: ActivateScreen("Feed Pump", 0)
   Button "Button_3" at 198,730 size 90x68; TextOn 'Fans'; TextOff 'Fans'
      on Click: ActivateScreen("ID FD Fan", 0)
   Button "Button_4" at 288,730 size 100x68; TextOn 'Stoker'; TextOff 'Stoker'
      on Click: ActivateScreen("Stoker", 0)
   Button "Button_6" at 516,730 size 89x68; TextOff 'Setup'
      on Click: ActivateScreen("Setup", 0)
   Button "Button_11" at 1164,730 size 114x68; TextOff 'Trends'
      on Click: ActivateScreen("Trend Steam", 0)
   Button "Button_18" at 387,730 size 129x68; TextOff 'Coal Handling'
      on Click: ActivateScreen("Coal Handling", 0)
   Button "Button_5" at 604,730 size 210x68; TextOff 'Coal & Blowdown Setup'
      on Click: ActivateScreen("Coal Setup", 0)
   Button "Button_19" at 814,730 size 140x68; TextOff 'Front/Rear Undergrate'
      on Click: ActivateScreen("Front Undergrate Damper", 0)
   Button "Button_20" at 954,730 size 100x68; TextOff 'Alarm Setup'
      on Click: ActivateScreen("Alarm Setup", 0)
   Button "Button_21" at 1054,730 size 110x68; TextOff 'Alarm History'
      on Click: ActivateScreen("Alarm History", 0)

screen "Coal Handling" 1280x800, template "Template_All"
   TextField "Text field_1" at 25,211 size 273x43; Text 'LH SWING CHUTE'
   TextField "Text field_2" at 357,211 size 277x43; Text 'RH SWING CHUTE'
   TextField "Text field_3" at 827,213 size 236x43; Text 'SINGLE BUCKET'
   TextField "Text field_14" at 808,214 size 15x22; Text 'E'
   TextField "Text field_15" at 790,253 size 36x37; Text 'LH'
   TextField "Text field_16" at 1040,254 size 40x37; Text 'RH'
   TextField "Text field_17" at 171,509 size 311x43; Text 'WET ASH CONVEYOR'
   TextField "Text field_18" at 72,470 size 18x22; Text 'O'
   TextField "Text field_19" at 507,111 size 292x50; Text 'COAL HANDLING'
   TextField "Text field_20" at 704,564 size 167x37; Text 'LH ON DELAY'
   TextField "Text field_21" at 704,618 size 171x37; Text 'RH ON DELAY'
   IOField "I/O field_1" at 933,559 size 127x44; FormatPattern 999
      ProcessValue <- "DATA_PARAMETER.DELAY_TIME_LH_BUCKET"
   IOField "I/O field_2" at 933,613 size 127x44; FormatPattern 999
      ProcessValue <- "DATA_PARAMETER.DELAY_TIME_RH_BUCKET"
   TextField "Text field_22" at 1082,563 size 46x37; Text 'Sec'
   TextField "Text field_23" at 1082,617 size 46x37; Text 'Sec'
   Switch "Switch_3" at 41,289 size 224x80; TextOn 'ON'; CaptionText 'Switch'; TextOff 'OFF'
      ProcessValue <- "DATA_SWITCH.SW_LHSWING"
      Appearance <- "DATA_STATUS.LH_SWING_STATUS"
   Switch "Switch_2" at 41,372 size 224x80; TextOn 'AUTO'; CaptionText 'Switch'; TextOff 'HAND'
      ProcessValue <- "DATA_SWITCH.AUTO_LHSWING"
      Appearance <- "DATA_SWITCH.AUTO_LHSWING"
   Switch "Switch_4" at 375,289 size 224x80; TextOn 'ON'; CaptionText 'Switch'; TextOff 'OFF'
      ProcessValue <- "DATA_SWITCH.SW_RHSWING"
      Appearance <- "DATA_STATUS.RH_SWING_STATUS"
   Switch "Switch_5" at 375,372 size 224x80; TextOn 'AUTO'; CaptionText 'Switch'; TextOff 'HAND'
      ProcessValue <- "DATA_SWITCH.AUTO_RHSWING"
      Appearance <- "DATA_SWITCH.AUTO_RHSWING"
   Switch "Switch_6" at 208,593 size 224x80; TextOn 'ON'; CaptionText 'Switch'; TextOff 'OFF'
      ProcessValue <- "DATA_SWITCH.SW_ASH_CONV"
      Appearance <- "DATA_STATUS.ASH_CONV_STATUS"
   Switch "Switch_7" at 700,289 size 224x80; TextOn 'AUTO'; CaptionText 'Switch'; TextOff 'HAND'
      ProcessValue <- "DATA_SWITCH.AUTO_LH_BUCKET"
      Appearance <- "DATA_SWITCH.AUTO_LH_BUCKET"
   Switch "Switch_10" at 952,289 size 224x80; TextOn 'AUTO'; CaptionText 'Switch'; TextOff 'HAND'
      ProcessValue <- "DATA_SWITCH.AUTO_RH_BUCKET"
      Appearance <- "DATA_SWITCH.AUTO_RH_BUCKET"
   Button "Button_12" at 700,371 size 224x80; TextOff 'UP'
      on Press: function_b14e0dd5("DATA_SWITCH.LH_HAND_BUCKET_UP", 0)
      Appearance <- "WORK_BIT.LH_SINGLE_BUCKET_UP"
   Button "Button_13" at 952,371 size 224x80; TextOff 'UP'
      on Press: function_b14e0dd5("DATA_SWITCH.RH_HAND_BUCKET_UP", 0)
      Appearance <- "WORK_BIT.RH_SINGLE_BUCKET_UP"
   Button "Button_14" at 700,453 size 224x80; TextOff 'DOWN'
      on Press: function_b14e0dd5("DATA_SWITCH.LH_HAND_BUCKET_DOWN", 0)
      Appearance <- "WORK_BIT.LH_SINGLE_BUCKET_DOWN"
   Button "Button_15" at 952,453 size 224x80; TextOff 'DOWN'
      on Press: function_b14e0dd5("DATA_SWITCH.RH_HAND_BUCKET_DOWN", 0)
      Appearance <- "WORK_BIT.RH_SINGLE_BUCKET_DOWN"
   Button "Button_1" at 0,730 size 98x68; TextOff 'Text'; PictureOn "Home_1"; PictureOff "Home_1"
      on Click: ActivateScreen("Home Screen", 0)
   Button "Button_2" at 98,730 size 100x68; TextOn 'Pumps'; TextOff 'Pumps'
      on Click: ActivateScreen("Feed Pump", 0)
   Button "Button_3" at 198,730 size 90x68; TextOn 'Fans'; TextOff 'Fans'
      on Click: ActivateScreen("ID FD Fan", 0)
   Button "Button_4" at 288,730 size 100x68; TextOn 'Stoker'; TextOff 'Stoker'
      on Click: ActivateScreen("Stoker", 0)
   Button "Button_6" at 516,730 size 89x68; TextOff 'Setup'
      on Click: ActivateScreen("Setup", 0)
   Button "Button_11" at 1164,730 size 114x68; TextOff 'Trends'
      on Click: ActivateScreen("Trend Steam", 0)
   Button "Button_18" at 387,730 size 129x68; TextOff 'Coal Handling'
      on Click: ActivateScreen("Coal Handling", 0)
   Button "Button_5" at 604,730 size 210x68; TextOff 'Coal & Blowdown Setup'
      on Click: ActivateScreen("Coal Setup", 0)
   Button "Button_19" at 814,730 size 140x68; TextOff 'Front/Rear Undergrate'
      on Click: ActivateScreen("Front Undergrate Damper", 0)
   Button "Button_20" at 954,730 size 100x68; TextOff 'Alarm Setup'
      on Click: ActivateScreen("Alarm Setup", 0)
   Button "Button_21" at 1054,730 size 110x68; TextOff 'Alarm History'
      on Click: ActivateScreen("Alarm History", 0)

screen "Setup" 1280x800, template "Template_All"
   on ClearScreen: function_f23ef4c9()
   TextField "Text field_2" at 124,187 size 156x34; Text 'O2 CONTROL'
   TextField "Text field_3" at 16,236 size 73x34; Text 'SP O2'
   TextField "Text field_14" at 16,289 size 168x34; Text 'MAX COMP O2'
   TextField "Text field_15" at 87,341 size 130x34; Text 'PID PUMPS'
   TextField "Text field_16" at 16,392 size 135x34; Text 'SETPOINTS'
   TextField "Text field_17" at 16,443 size 63x34; Text 'GAIN'
   TextField "Text field_18" at 16,494 size 29x34; Text 'TI'
   TextField "Text field_19" at 16,548 size 37x34; Text 'TD'
   TextField "Text field_20" at 16,601 size 130x34; Text 'LSP PUMPS'
   TextField "Text field_21" at 16,653 size 128x34; Text 'MAX FLOW'
   IOField "I/O field_1" at 220,231 size 119x44; FormatPattern 99.9
      ProcessValue <- "DATA_PARAMETER.SP_O2"
   IOField "I/O field_2" at 220,284 size 119x44; FormatPattern 999
      ProcessValue <- "DATA_PARAMETER.MAX_PERC_O2"
   IOField "I/O field_3" at 220,387 size 119x44; FormatPattern 999.9
      ProcessValue <- "DATA_PARAMETER.SP_WATER_LEVEL"
   IOField "I/O field_4" at 220,438 size 119x44; Authorization "Operate"; FormatPattern 999.9
      ProcessValue <- "DATA_PARAMETER.GAIN_PUMPS"
   IOField "I/O field_5" at 220,490 size 119x44; Authorization "Operate"; FormatPattern 999.9
      ProcessValue <- "DATA_PARAMETER.TI_PUMPS"
   IOField "I/O field_6" at 220,543 size 119x44; Authorization "Operate"; FormatPattern 999.9
      ProcessValue <- "DATA_PARAMETER.TD_PUMPS"
   IOField "I/O field_7" at 220,596 size 119x44; Authorization "Operate"; FormatPattern 999.9
      ProcessValue <- "DATA_PARAMETER.LSP_PUMPS"
   IOField "I/O field_8" at 220,648 size 119x44; Authorization "Operate"; FormatPattern 999.9
      ProcessValue <- "DATA_PARAMETER.MAX_FLOWRATE"
   TextField "Text field_22" at 359,236 size 29x34; Text '%'
   TextField "Text field_23" at 359,289 size 29x34; Text '%'
   TextField "Text field_24" at 359,392 size 29x34; Text '%'
   TextField "Text field_25" at 344,494 size 44x34; Text 'Sec'
   TextField "Text field_26" at 351,548 size 37x34; Text 'ms'
   TextField "Text field_27" at 355,601 size 33x34; Text 'Hz'
   TextField "Text field_28" at 324,653 size 62x34; Text 'm³/h'
   TextField "Text field_29" at 484,187 size 169x34; Text 'FD FAN SETUP'
   TextField "Text field_30" at 431,236 size 135x34; Text 'SETPOINTS'
   IOField "I/O field_9" at 626,231 size 119x44; FormatPattern 999.9
      ProcessValue <- "SP_FD_FAN"
   TextField "Text field_31" at 765,236 size 41x34; Text 'bar'
   TextField "Text field_32" at 431,289 size 63x34; Text 'GAIN'
   TextField "Text field_33" at 431,341 size 29x34; Text 'TI'
   TextField "Text field_34" at 431,392 size 37x34; Text 'TD'
   IOField "I/O field_10" at 626,284 size 119x44; FormatPattern 999.9
      ProcessValue <- "DATA_PARAMETER.GAIN_FD"
   IOField "I/O field_11" at 626,336 size 119x44; FormatPattern 999.9
      ProcessValue <- "DATA_PARAMETER.TI_FD"
   IOField "I/O field_12" at 626,387 size 119x44; FormatPattern 999.9
      ProcessValue <- "PID_STOKER.TD"
   TextField "Text field_35" at 765,341 size 44x34; Text 'Sec'
   TextField "Text field_36" at 765,392 size 37x34; Text 'ms'
   TextField "Text field_37" at 431,443 size 112x34; Text 'LSP LHFD'
   TextField "Text field_38" at 431,494 size 117x34; Text 'HSP LHFD'
   TextField "Text field_39" at 431,548 size 116x34; Text 'LSP RHFD'
   TextField "Text field_40" at 431,601 size 121x34; Text 'HSP RHFD'
   TextField "Text field_41" at 431,653 size 132x34; Text 'LSP ID FAN'
   IOField "I/O field_13" at 626,438 size 119x44; FormatPattern 99.9
      ProcessValue <- "DATA_PARAMETER.LSP_LHFD_FAN"
   TextField "Text field_42" at 765,443 size 33x34; Text 'Hz'
   IOField "I/O field_14" at 626,491 size 119x44; FormatPattern 99.9
      ProcessValue <- "DATA_PARAMETER.HSP_LHFD_FAN"
   TextField "Text field_43" at 765,494 size 33x34; Text 'Hz'
   IOField "I/O field_15" at 626,543 size 119x44; FormatPattern 99.9
      ProcessValue <- "DATA_PARAMETER.LSP_RHFD_FAN"
   TextField "Text field_44" at 765,548 size 33x34; Text 'Hz'
   IOField "I/O field_16" at 626,596 size 119x44; FormatPattern 99.9
      ProcessValue <- "DATA_PARAMETER.HSP_RHFD_FAN"
   TextField "Text field_45" at 765,601 size 33x34; Text 'Hz'
   IOField "I/O field_17" at 626,648 size 119x44; FormatPattern 99.9
      ProcessValue <- "DATA_PARAMETER.LSP_ID_FAN"
   TextField "Text field_46" at 765,653 size 33x34; Text 'Hz'
   TextField "Text field_47" at 850,236 size 135x34; Text 'SETPOINTS'
   IOField "I/O field_18" at 1079,236 size 118x35; FormatPattern 999.9
      ProcessValue <- "PID_STROKER_SETPOINT"
   TextField "Text field_48" at 1209,236 size 41x34; Text 'bar'
   TextField "Text field_49" at 850,289 size 63x34; Text 'GAIN'
   TextField "Text field_50" at 850,341 size 29x34; Text 'TI'
   TextField "Text field_51" at 850,392 size 37x34; Text 'TD'
   IOField "I/O field_19" at 1079,284 size 119x44; FormatPattern 999.9
      ProcessValue <- "PID_STOKER.GAIN"
   IOField "I/O field_20" at 1079,336 size 119x44; FormatPattern 999.9
      ProcessValue <- "PID_STOKER.TI"
   IOField "I/O field_21" at 1079,387 size 119x44; FormatPattern 999.9
      ProcessValue <- "PID_STOKER.TD"
   TextField "Text field_52" at 1209,341 size 44x34; Text 'Sec'
   TextField "Text field_53" at 1209,392 size 37x34; Text 'ms'
   TextField "Text field_54" at 850,443 size 182x34; Text 'LSP LH STOKER'
   TextField "Text field_55" at 850,494 size 187x34; Text 'HSP LH STOKER'
   TextField "Text field_56" at 850,548 size 186x34; Text 'LSP RH STOKER'
   IOField "I/O field_22" at 1079,438 size 119x44; FormatPattern 99.9
      ProcessValue <- "DATA_PARAMETER.LSP_LH_STOKER"
   TextField "Text field_57" at 1209,443 size 33x34; Text 'Hz'
   IOField "I/O field_23" at 1079,490 size 119x44; FormatPattern 99.9
      ProcessValue <- "DATA_PARAMETER.HSP_LH_STOKER"
   TextField "Text field_58" at 1209,494 size 33x34; Text 'Hz'
   TextField "Text field_59" at 850,601 size 191x34; Text 'HSP RH STOKER'
   TextField "Text field_60" at 850,653 size 137x34; Text 'HSP ID FAN'
   IOField "I/O field_24" at 1079,596 size 119x44; FormatPattern 99.9
      ProcessValue <- "DATA_PARAMETER.HSP_RH_STOKER"
   TextField "Text field_61" at 1209,601 size 33x34; Text 'Hz'
   IOField "I/O field_25" at 1079,648 size 119x44; FormatPattern 999.9
      ProcessValue <- "DATA_PARAMETER.HSP_ID_FAN"
   TextField "Text field_62" at 1209,653 size 33x34; Text 'Hz'
   IOField "I/O field_26" at 1079,543 size 119x44; FormatPattern 99.9
      ProcessValue <- "DATA_PARAMETER.LSP_RH_STOKER"
   TextField "Text field_63" at 1209,548 size 33x34; Text 'Hz'
   TextField "Text field_64" at 453,112 size 335x50; Text 'PARAMETER SETUP'
   TextField "Text field_65" at 930,187 size 145x34; Text 'PID STOKER'
   Button "Button_1" at 0,730 size 98x68; TextOff 'Text'; PictureOn "Home_1"; PictureOff "Home_1"
      on Click: ActivateScreen("Home Screen", 0)
   Button "Button_2" at 98,730 size 100x68; TextOn 'Pumps'; TextOff 'Pumps'
      on Click: ActivateScreen("Feed Pump", 0)
   Button "Button_3" at 198,730 size 90x68; TextOn 'Fans'; TextOff 'Fans'
      on Click: ActivateScreen("ID FD Fan", 0)
   Button "Button_4" at 288,730 size 100x68; TextOn 'Stoker'; TextOff 'Stoker'
      on Click: ActivateScreen("Stoker", 0)
   Button "Button_6" at 516,730 size 89x68; TextOff 'Setup'
      on Click: ActivateScreen("Setup", 0)
   Button "Button_11" at 1164,730 size 114x68; TextOff 'Trends'
      on Click: ActivateScreen("Trend Steam", 0)
   Button "Button_5" at 387,730 size 129x68; TextOff 'Coal Handling'
      on Click: ActivateScreen("Coal Handling", 0)
   Button "Button_7" at 604,730 size 210x68; TextOff 'Coal & Blowdown Setup'
      on Click: ActivateScreen("Coal Setup", 0)
   Button "Button_8" at 814,730 size 140x68; TextOff 'Front/Rear Undergrate'
      on Click: ActivateScreen("Front Undergrate Damper", 0)
   Button "Button_20" at 954,730 size 100x68; TextOff 'Alarm Setup'
      on Click: ActivateScreen("Alarm Setup", 0)
   Button "Button_21" at 1054,730 size 110x68; TextOff 'Alarm History'
      on Click: ActivateScreen("Alarm History", 0)
   Button "Button_9" at 305,334 size 98x48; TextOff 'TREND'
      on Click: ActivateScreen("Trend PID Pump", 0)
   Button "Button_10" at 726,180 size 98x48; TextOff 'TREND'
      on Click: ActivateScreen("Trend PID FD Fan", 0)
   Button "Button_12" at 1172,180 size 98x48; TextOff 'TREND'
      on Click: ActivateScreen("Trend PID Stoker", 0)
   Button "Button_13" at 515,730 size 91x68; TextOff 'Text'; Authorization "User administration"
      on Click: ActivateScreen("AI Min Max Setting", 0)

screen "Coal Setup" 1280x800, template "Template_All"
   TextField "Text field_1" at 530,111 size 219x50; Text 'COAL SETUP'
   TextField "Text field_16" at 129,285 size 172x37; Text 'COAL HEIGHT'
   TextField "Text field_2" at 135,337 size 113x37; Text 'DENSITY'
   TextField "Text field_3" at 657,285 size 172x37; Text 'COAL HEIGHT'
   TextField "Text field_14" at 665,337 size 113x37; Text 'DENSITY'
   TextField "Text field_15" at 500,286 size 51x37; Text 'mm'
   TextField "Text field_17" at 1022,285 size 51x37; Text 'mm'
   TextField "Text field_18" at 240,183 size 195x37; Text 'LH COAL SETUP'
   TextField "Text field_19" at 755,184 size 199x37; Text 'RH COAL SETUP'
   IOField "I/O field_1" at 349,285 size 138x42; FormatPattern 999.9
      ProcessValue <- "DATA_PARAMETER.LH_COAL_HEIGHT"
   IOField "I/O field_2" at 349,335 size 138x42; FormatPattern 9.999
      ProcessValue <- "DATA_PARAMETER.LH_DENSITY"
   IOField "I/O field_3" at 874,284 size 138x42; FormatPattern 999.9
      ProcessValue <- "DATA_PARAMETER.RH_COAL_HEIGHT"
   IOField "I/O field_4" at 874,335 size 138x42; FormatPattern 9.999
      ProcessValue <- "DATA_PARAMETER.RH_DENSITY"
   Button "Button_1" at 0,730 size 98x68; TextOff 'Text'; PictureOn "Home_1"; PictureOff "Home_1"
      on Click: ActivateScreen("Home Screen", 0)
   Button "Button_2" at 98,730 size 100x68; TextOn 'Pumps'; TextOff 'Pumps'
      on Click: ActivateScreen("Feed Pump", 0)
   Button "Button_3" at 198,730 size 90x68; TextOn 'Fans'; TextOff 'Fans'
      on Click: ActivateScreen("ID FD Fan", 0)
   Button "Button_4" at 288,730 size 100x68; TextOn 'Stoker'; TextOff 'Stoker'
      on Click: ActivateScreen("Stoker", 0)
   Button "Button_6" at 516,730 size 89x68; TextOff 'Setup'
      on Click: ActivateScreen("Setup", 0)
   Button "Button_11" at 1164,730 size 114x68; TextOff 'Trends'
      on Click: ActivateScreen("Trend Steam", 0)
   Button "Button_18" at 387,730 size 129x68; TextOff 'Coal Handling'
      on Click: ActivateScreen("Coal Handling", 0)
   Button "Button_5" at 604,730 size 210x68; TextOff 'Blowdown Setup'
      on Click: ActivateScreen("Blowdown Setup", 0)
   Button "Button_19" at 814,730 size 140x68; TextOff 'Front/Rear Undergrate'
      on Click: ActivateScreen("Front Undergrate Damper", 0)
   Button "Button_20" at 954,730 size 100x68; TextOff 'Alarm Setup'
      on Click: ActivateScreen("Alarm Setup", 0)
   Button "Button_21" at 1054,730 size 110x68; TextOff 'Alarm History'
      on Click: ActivateScreen("Alarm History", 0)

screen "Blowdown Setup" 1280x800, template "Template_All"
   TextField "Text field_1" at 466,112 size 341x50; Text 'BLOWDOWN SETUP'
   TextField "Text field_2" at 464,235 size 122x37; Text 'OFF TIME'
   TextField "Text field_3" at 464,286 size 136x37; Text 'OFF PULSE'
   TextField "Text field_14" at 464,337 size 126x37; Text 'ON PULSE'
   TextField "Text field_15" at 464,389 size 114x37; Text 'PERIODE'
   IOField "I/O field_1" at 652,232 size 121x43; FormatPattern 999
      ProcessValue <- "DATA_PARAMETER.OFF_TIME_BLOWDOWN"
   IOField "I/O field_2" at 652,282 size 121x43; FormatPattern 999
      ProcessValue <- "DATA_PARAMETER.OFF_PULSE_BLOWDOWN"
   IOField "I/O field_3" at 652,333 size 121x43; FormatPattern 999
      ProcessValue <- "DATA_PARAMETER.ON_PULSE_BLOWDOWN"
   IOField "I/O field_4" at 652,386 size 121x43; FormatPattern 999
      ProcessValue <- "DATA_PARAMETER.PERIODE"
   TextField "Text field_16" at 773,235 size 49x37; Text 'min'
   TextField "Text field_17" at 773,286 size 43x37; Text 'sec'
   TextField "Text field_18" at 773,337 size 43x37; Text 'sec'
   TextField "Text field_19" at 773,388 size 69x37; Text 'times'
   Switch "Switch_1" at 524,444 size 226x86; TextOn 'AUTO'; CaptionText 'Switch'; TextOff 'HAND'
      ProcessValue <- "Hand/Auto_Blowdown"
      Appearance <- "Hand/Auto_Blowdown"
   Button "Button_1" at 0,730 size 98x68; TextOff 'Text'; PictureOn "Home_1"; PictureOff "Home_1"
      on Click: ActivateScreen("Home Screen", 0)
   Button "Button_2" at 98,730 size 100x68; TextOn 'Pumps'; TextOff 'Pumps'
      on Click: ActivateScreen("Feed Pump", 0)
   Button "Button_3" at 198,730 size 90x68; TextOn 'Fans'; TextOff 'Fans'
      on Click: ActivateScreen("ID FD Fan", 0)
   Button "Button_4" at 288,730 size 100x68; TextOn 'Stoker'; TextOff 'Stoker'
      on Click: ActivateScreen("Stoker", 0)
   Button "Button_6" at 516,730 size 89x68; TextOff 'Setup'
      on Click: ActivateScreen("Setup", 0)
   Button "Button_11" at 1164,730 size 114x68; TextOff 'Trends'
      on Click: ActivateScreen("Trend Steam", 0)
   Button "Button_18" at 387,730 size 129x68; TextOff 'Coal Handling'
      on Click: ActivateScreen("Coal Handling", 0)
   Button "Button_5" at 604,730 size 210x68; TextOff 'Coal & Blowdown Setup'
      on Click: ActivateScreen("Coal Setup", 0)
   Button "Button_19" at 814,730 size 140x68; TextOff 'Front/Rear Undergrate'
      on Click: ActivateScreen("Front Undergrate Damper", 0)
   Button "Button_20" at 954,730 size 100x68; TextOff 'Alarm Setup'
      on Click: ActivateScreen("Alarm Setup", 0)
   Button "Button_21" at 1054,730 size 110x68; TextOff 'Alarm History'
      on Click: ActivateScreen("Alarm History", 0)
   Switch "Switch_3" at 524,532 size 226x86; TextOn 'ON BLOWDOWN'; CaptionText 'Switch'; TextOff 'OFF BLOWDOWN'
      Appearance <- "PB_BLOWDOWN"
      ProcessValue <- "PB_BLOWDOWN"
      Visibility <- "Hand/Auto_Blowdown"

screen "Rear Undergrate Damper" 1280x800, template "Template_All"
   Button "Button_12" at 209,262 size 221x81; TextOn 'OPEN'; TextOff 'OPEN'
      on Press: function_b14e0dd5("DATA_SWITCH.HAND_LH_REAR_UND_OPEN", 0)
      Appearance <- "DATA_SWITCH.HAND_LH_REAR_UND_OPEN"
   Button "Button_13" at 209,343 size 221x81; TextOn 'CLOSE'; TextOff 'CLOSE'
      on Press: function_b14e0dd5("DATA_SWITCH.HAND_LH_REAR_UND_CLOSE", 0)
      Appearance <- "DATA_SWITCH.HAND_LH_REAR_UND_CLOSE"
   Button "Button_14" at 818,262 size 221x81; TextOn 'OPEN'; TextOff 'OPEN'
      on Press: function_b14e0dd5("DATA_SWITCH.HAND_RH_REAR_UND_OPEN", 0)
      Appearance <- "DATA_SWITCH.HAND_RH_REAR_UND_OPEN"
   Button "Button_15" at 818,343 size 221x81; TextOn 'CLOSE'; TextOff 'CLOSE'
      on Press: function_b14e0dd5("DATA_SWITCH.HAND_RH_REAR_UND_CLOSE", 0)
      Appearance <- "DATA_SWITCH.HAND_RH_REAR_UND_CLOSE"
   TextField "Text field_1" at 177,184 size 285x37; Text 'LH REAR UNDERGRATE'
   TextField "Text field_2" at 784,183 size 289x37; Text 'RH REAR UNDERGRATE'
   TextField "Text field_3" at 308,111 size 623x50; Text 'REAR UNDERGRATE DAMPER SETUP'
   TextField "Text field_14" at 94,530 size 153x34; Text 'LH FD SPEED'
   TextField "Text field_15" at 94,578 size 215x34; Text 'LH REAR UND POS'
   TextField "Text field_16" at 734,529 size 157x34; Text 'RH FD SPEED'
   TextField "Text field_17" at 734,577 size 219x34; Text 'RH REAR UND POS'
   IOField "I/O field_1" at 356,531 size 132x36; FormatPattern 999.9
      ProcessValue <- "LHFD_SCALING.Value"
   IOField "I/O field_2" at 356,578 size 132x36; FormatPattern 999.9
      ProcessValue <- "ANALOG_DISPLAY.LH_REAR_UND_POS"
   IOField "I/O field_3" at 1000,532 size 132x36; FormatPattern 999.9
      ProcessValue <- "RH_FD_SCALING.Value"
   IOField "I/O field_4" at 1000,578 size 132x36; FormatPattern 999.9
      ProcessValue <- "ANALOG_DISPLAY.RH_REAR_UND_POS"
   TextField "Text field_18" at 488,531 size 29x34; Text '%'
   TextField "Text field_19" at 1125,530 size 29x34; Text '%'
   TextField "Text field_20" at 488,578 size 100x34; Text '% OPEN'
   TextField "Text field_21" at 1125,578 size 100x34; Text '% OPEN'
   Button "Button_1" at 0,730 size 98x68; TextOff 'Text'; PictureOn "Home_1"; PictureOff "Home_1"
      on Click: ActivateScreen("Home Screen", 0)
   Button "Button_2" at 98,730 size 100x68; TextOn 'Pumps'; TextOff 'Pumps'
      on Click: ActivateScreen("Feed Pump", 0)
   Button "Button_3" at 198,730 size 90x68; TextOn 'Fans'; TextOff 'Fans'
      on Click: ActivateScreen("ID FD Fan", 0)
   Button "Button_4" at 288,730 size 100x68; TextOn 'Stoker'; TextOff 'Stoker'
      on Click: ActivateScreen("Stoker", 0)
   Button "Button_6" at 516,730 size 89x68; TextOff 'Setup'
      on Click: ActivateScreen("Setup", 0)
   Button "Button_11" at 1164,730 size 114x68; TextOff 'Trends'
      on Click: ActivateScreen("Trend Steam", 0)
   Button "Button_5" at 387,730 size 129x68; TextOff 'Coal Handling'
      on Click: ActivateScreen("Coal Handling", 0)
   Button "Button_7" at 604,730 size 210x68; TextOff 'Coal & Blowdown Setup'
      on Click: ActivateScreen("Coal Setup", 0)
   Button "Button_8" at 814,730 size 140x68; TextOff 'Front/Rear Undergrate'
      on Click: ActivateScreen("Front Undergrate Damper", 0)
   Button "Button_20" at 954,730 size 100x68; TextOff 'Alarm Setup'
      on Click: ActivateScreen("Alarm Setup", 0)
   Button "Button_21" at 1054,730 size 110x68; TextOff 'Alarm History'
      on Click: ActivateScreen("Alarm History", 0)

screen "Front Undergrate Damper" 1280x800, template "Template_All"
   TextField "Text field_3" at 318,107 size 649x50; Text 'FRONT UNDERGRATE DAMPER SETUP'
   TextField "Text field_1" at 192,167 size 304x37; Text 'LH FRONT UNDERGRATE'
   TextField "Text field_2" at 790,167 size 308x37; Text 'RH FRONT UNDERGRATE'
   TextField "Text field_14" at 34,491 size 162x37; Text 'LH FD SPEED'
   TextField "Text field_15" at 34,542 size 247x37; Text 'LH FRONT UND POS'
   TextField "Text field_16" at 34,595 size 224x37; Text 'LH OFFSET SETUP'
   TextField "Text field_17" at 693,491 size 166x37; Text 'RH FD SPEED'
   TextField "Text field_18" at 693,542 size 251x37; Text 'RH FRONT UND POS'
   TextField "Text field_19" at 693,595 size 228x37; Text 'RH OFFSET SETUP'
   TextField "Text field_20" at 473,489 size 31x37; Text '%'
   TextField "Text field_21" at 473,540 size 106x37; Text '% OPEN'
   TextField "Text field_22" at 1131,492 size 31x37; Text '%'
   TextField "Text field_23" at 1131,543 size 106x37; Text '% OPEN'
   TextField "Text field_24" at 1131,596 size 31x37; Text '%'
   TextField "Text field_25" at 473,596 size 31x37; Text '%'
   IOField "I/O field_1" at 338,540 size 122x40; FormatPattern 999.9
      ProcessValue <- "ANALOG_DISPLAY.LH_FRONT_UND_POS"
   IOField "I/O field_2" at 338,491 size 122x40; FormatPattern 999.9
      ProcessValue <- "LHFD_SCALING.Value"
   IOField "I/O field_3" at 338,592 size 122x40; FormatPattern 999
      ProcessValue <- "DATA_PARAMETER.LH_OFFSET"
   IOField "I/O field_4" at 993,540 size 122x40; FormatPattern 999.9
      ProcessValue <- "ANALOG_DISPLAY.RH_FRONT_UND_POS"
   IOField "I/O field_5" at 993,491 size 122x40; FormatPattern 999.9
      ProcessValue <- "RH_FD_SCALING.Value"
   IOField "I/O field_6" at 993,592 size 122x40; FormatPattern 999
      ProcessValue <- "DATA_PARAMETER.RH_OFFSET"
   Button "Button_1" at 0,730 size 98x68; TextOff 'Text'; PictureOn "Home_1"; PictureOff "Home_1"
      on Click: ActivateScreen("Home Screen", 0)
   Button "Button_2" at 98,730 size 100x68; TextOn 'Pumps'; TextOff 'Pumps'
      on Click: ActivateScreen("Feed Pump", 0)
   Button "Button_3" at 198,730 size 90x68; TextOn 'Fans'; TextOff 'Fans'
      on Click: ActivateScreen("ID FD Fan", 0)
   Button "Button_4" at 288,730 size 100x68; TextOn 'Stoker'; TextOff 'Stoker'
      on Click: ActivateScreen("Stoker", 0)
   Button "Button_6" at 516,730 size 89x68; TextOff 'Setup'
      on Click: ActivateScreen("Setup", 0)
   Button "Button_11" at 1164,730 size 114x68; TextOff 'Trends'
      on Click: ActivateScreen("Trend Steam", 0)
   Button "Button_18" at 387,730 size 129x68; TextOff 'Coal Handling'
      on Click: ActivateScreen("Coal Handling", 0)
   Button "Button_5" at 604,730 size 210x68; TextOff 'Coal & Blowdown Setup'
      on Click: ActivateScreen("Coal Setup", 0)
   Button "Button_19" at 814,730 size 140x68; TextOff 'Rear Undergrate'
      on Click: ActivateScreen("Rear Undergrate Damper", 0)
   Button "Button_20" at 954,730 size 100x68; TextOff 'Alarm Setup'
      on Click: ActivateScreen("Alarm Setup", 0)
   Button "Button_21" at 1054,730 size 110x68; TextOff 'Alarm History'
      on Click: ActivateScreen("Alarm History", 0)
   Switch "Switch_1" at 231,224 size 225x81; TextOn 'AUTO'; CaptionText 'Switch'; TextOff 'HAND'
      ProcessValue <- "DATA_SWITCH.AUTO_LHFRONT_UND_SW"
      Appearance <- "DATA_SWITCH.AUTO_LHFRONT_UND_SW"
   Switch "Switch_2" at 831,224 size 225x81; TextOn 'AUTO'; CaptionText 'Switch'; TextOff 'HAND'
      ProcessValue <- "DATA_SWITCH.AUTO_RHFRONT_UND_SW"
      Appearance <- "DATA_SWITCH.AUTO_RHFRONT_UND_SW"
   Button "Button_10" at 231,306 size 225x81; TextOff 'OPEN'
      on Press: function_b14e0dd5("DATA_SWITCH.HAND_LH_FRONT_UND_OPEN", 0)
      Appearance <- "DATA_SWITCH.HAND_LH_FRONT_UND_OPEN"
   Button "Button_7" at 231,388 size 225x81; TextOff 'CLOSED'
      on Press: function_b14e0dd5("DATA_SWITCH.HAND_LH_FRONT_UND_CLOSE", 0)
      Appearance <- "DATA_SWITCH.HAND_LH_FRONT_UND_CLOSE"
   Button "Button_8" at 831,306 size 225x81; TextOff 'OPEN'
      on Press: function_b14e0dd5("DATA_SWITCH.HAND_RH_FRONT_UND_OPEN", 0)
      Appearance <- "DATA_SWITCH.HAND_RH_FRONT_UND_OPEN"
   Button "Button_9" at 831,388 size 225x81; TextOff 'CLOSED'
      on Press: function_b14e0dd5("DATA_SWITCH.HAND_RH_FRONT_UND_CLOSE", 0)
      Appearance <- "DATA_SWITCH.HAND_RH_FRONT_UND_CLOSE"

screen "Alarm Setup" 1280x800, template "Template_All"
   TextField "Text field_17" at 108,184 size 173x37; Text 'WATER LEVEL'
   TextField "Text field_1" at 515,183 size 213x37; Text 'BURNBACK TEMP'
   TextField "Text field_2" at 941,184 size 223x37; Text 'STEAM PRESSURE'
   TextField "Text field_3" at 520,110 size 245x50; Text 'ALARM SETUP'
   TextField "Text field_14" at 8,292 size 218x37; Text 'LW PREWARNING'
   TextField "Text field_15" at 12,340 size 165x37; Text 'HIGH WATER'
   TextField "Text field_16" at 466,291 size 215x37; Text 'SP LH BURNBACK'
   TextField "Text field_18" at 466,340 size 219x37; Text 'SP RH BURNBACK'
   TextField "Text field_19" at 935,291 size 99x37; Text 'SP LOW'
   TextField "Text field_20" at 934,340 size 107x37; Text 'SP HIGH'
   IOField "I/O field_1" at 270,285 size 106x45; FormatPattern 999.9
      ProcessValue <- "WTR_LEVEL_SCALING.SP_L"
   IOField "I/O field_2" at 274,335 size 102x45; FormatPattern 999.9
      ProcessValue <- "WTR_LEVEL_SCALING.SP_H"
   IOField "I/O field_3" at 710,285 size 108x45; FormatPattern 999.9
      ProcessValue <- "LH_BURNBACK_TEMP.SP_H"
   IOField "I/O field_5" at 1064,286 size 102x45; FormatPattern 999.9
      ProcessValue <- "STEAM_PRESS.SP_L"
   IOField "I/O field_6" at 1064,337 size 102x45; FormatPattern 999.9
      ProcessValue <- "STEAM_PRESS.SP_H"
   TextField "Text field_21" at 377,291 size 31x37; Text '%'
   TextField "Text field_22" at 376,340 size 31x37; Text '%'
   TextField "Text field_23" at 830,290 size 21x37; Text 'C'
   TextField "Text field_24" at 830,342 size 21x37; Text 'C'
   TextField "Text field_25" at 1175,291 size 44x37; Text 'bar'
   TextField "Text field_26" at 1176,337 size 44x37; Text 'bar'
   IOField "I/O field_4" at 716,336 size 102x45; FormatPattern 999.9
      ProcessValue <- "RH_BURNBACK_TEMP.SP_H"
   Button "Button_1" at 0,730 size 98x68; TextOff 'Text'; PictureOn "Home_1"; PictureOff "Home_1"
      on Click: ActivateScreen("Home Screen", 0)
   Button "Button_2" at 98,730 size 100x68; TextOn 'Pumps'; TextOff 'Pumps'
      on Click: ActivateScreen("Feed Pump", 0)
   Button "Button_3" at 198,730 size 90x68; TextOn 'Fans'; TextOff 'Fans'
      on Click: ActivateScreen("ID FD Fan", 0)
   Button "Button_4" at 288,730 size 100x68; TextOn 'Stoker'; TextOff 'Stoker'
      on Click: ActivateScreen("Stoker", 0)
   Button "Button_6" at 516,730 size 89x68; TextOff 'Setup'
      on Click: ActivateScreen("Setup", 0)
   Button "Button_11" at 1164,730 size 114x68; TextOff 'Trends'
      on Click: ActivateScreen("Trend Steam", 0)
   Button "Button_18" at 387,730 size 129x68; TextOff 'Coal Handling'
      on Click: ActivateScreen("Coal Handling", 0)
   Button "Button_5" at 604,730 size 210x68; TextOff 'Coal & Blowdown Setup'
      on Click: ActivateScreen("Coal Setup", 0)
   Button "Button_19" at 814,730 size 140x68; TextOff 'Front/Rear Undergrate'
      on Click: ActivateScreen("Front Undergrate Damper", 0)
   Button "Button_20" at 954,730 size 100x68; TextOff 'Alarm Setup'
      on Click: ActivateScreen("Alarm Setup", 0)
   Button "Button_21" at 1054,730 size 110x68; TextOff 'Alarm History'
      on Click: ActivateScreen("Alarm History", 0)

